LIN {X 0,Y 192.714,Z 301.29,A -85,B 0,C 180,E1 -21855.206,E2 -21855.206} C_VEL
LIN {X 0,Y 192.91,Z 301.267,A -85,B 0,C 180,E1 -21859.549,E2 -21859.549} C_VEL
LIN {X 0,Y 193.003,Z 301.257,A -85,B 0,C 180,E1 -21861.621,E2 -21861.621} C_VEL
LIN {X 0,Y 193.24,Z 301.226,A -85,B 0,C 180,E1 -21867.912,E2 -21867.912} C_VEL
LIN {X 0,Y 193.401,Z 301.208,A -85,B 0,C 180,E1 -21869.996,E2 -21869.996} C_VEL
LIN {X 0,Y 192.941,Z 301.26,A -85,B 0,C 180,E1 -21874.174,E2 -21874.174} C_VEL
LIN {X 0,Y 193,Z 301.258,A -85,B 0,C 180,E1 -21878.372,E2 -21878.372} C_VEL
LIN {X 0,Y 192.755,Z 301.282,A -85,B 0,C 180,E1 -21882.633,E2 -21882.633} C_VEL
LIN {X 0,Y 192.704,Z 301.293,A -85,B 0,C 180,E1 -21886.96,E2 -21886.96} C_VEL
LIN {X 0,Y 192.567,Z 301.305,A -85,B 0,C 180,E1 -21891.401,E2 -21891.401} C_VEL
LIN {X 0,Y 192.6,Z 301.303,A -85,B 0,C 180,E1 -21894.214,E2 -21894.214} C_VEL
LIN {X 0,Y 192.604,Z 301.305,A -85,B 0,C 180,E1 -21898.895,E2 -21898.895} C_VEL
LIN {X 0,Y 192.556,Z 301.311,A -85,B 0,C 180,E1 -21903.189,E2 -21903.189} C_VEL
LIN {X 0,Y 192.57,Z 301.307,A -85,B 0,C 180,E1 -21908.342,E2 -21908.342} C_VEL
LIN {X 0,Y 192.587,Z 301.308,A -85,B 0,C 180,E1 -21913.145,E2 -21913.145} C_VEL
LIN {X 0,Y 192.582,Z 301.308,A -85,B 0,C 180,E1 -21916.869,E2 -21916.869} C_VEL
LIN {X 0,Y 192.564,Z 301.311,A -85,B 0,C 180,E1 -21921.667,E2 -21921.667} C_VEL
LIN {X 0,Y 192.564,Z 301.308,A -85,B 0,C 180,E1 -21926.822,E2 -21926.822} C_VEL
LIN {X 0,Y 192.629,Z 301.303,A -85,B 0,C 180,E1 -21931.7,E2 -21931.7} C_VEL
LIN {X 0,Y 192.655,Z 301.295,A -85,B 0,C 180,E1 -21936.355,E2 -21936.355} C_VEL
LIN {X 0,Y 192.672,Z 301.296,A -85,B 0,C 180,E1 -21941.498,E2 -21941.498} C_VEL
LIN {X 0,Y 192.716,Z 301.288,A -85,B 0,C 180,E1 -21945.222,E2 -21945.222} C_VEL
LIN {X 0,Y 192.925,Z 301.264,A -85,B 0,C 180,E1 -21949.577,E2 -21949.577} C_VEL
LIN {X 0,Y 192.954,Z 301.26,A -85,B 0,C 180,E1 -21953.738,E2 -21953.738} C_VEL
LIN {X 0,Y 193.218,Z 301.227,A -85,B 0,C 180,E1 -21957.926,E2 -21957.926} C_VEL
LIN {X 0,Y 193.4,Z 301.206,A -85,B 0,C 180,E1 -21960.01,E2 -21960.01} C_VEL
LIN {X 0,Y 192.932,Z 301.261,A -85,B 0,C 180,E1 -21964.188,E2 -21964.188} C_VEL
LIN {X 0,Y 193.012,Z 301.254,A -85,B 0,C 180,E1 -21968.385,E2 -21968.385} C_VEL
LIN {X 0,Y 192.769,Z 301.283,A -85,B 0,C 180,E1 -21972.646,E2 -21972.646} C_VEL
LIN {X 0,Y 192.691,Z 301.294,A -85,B 0,C 180,E1 -21978.518,E2 -21978.518} C_VEL
LIN {X 0,Y 192.61,Z 301.301,A -85,B 0,C 180,E1 -21984.198,E2 -21984.198} C_VEL
LIN {X 0,Y 192.602,Z 301.305,A -85,B 0,C 180,E1 -21988.874,E2 -21988.874} C_VEL
LIN {X 0,Y 192.598,Z 301.304,A -85,B 0,C 180,E1 -21993.196,E2 -21993.196} C_VEL
LIN {X 0,Y 192.547,Z 301.31,A -85,B 0,C 180,E1 -21998.364,E2 -21998.364} C_VEL
LIN {X 0,Y 192.492,Z 301.317,A -85,B 0,C 180,E1 -22003.102,E2 -22003.102} C_VEL
LIN {X 0,Y 192.493,Z 301.317,A -85,B 0,C 180,E1 -22006.916,E2 -22006.916} C_VEL
LIN {X 0,Y 192.553,Z 301.31,A -85,B 0,C 180,E1 -22011.654,E2 -22011.654} C_VEL
LIN {X 0,Y 192.608,Z 301.301,A -85,B 0,C 180,E1 -22016.821,E2 -22016.821} C_VEL
LIN {X 0,Y 192.73,Z 301.288,A -85,B 0,C 180,E1 -22021.707,E2 -22021.707} C_VEL
LIN {X 0,Y 193.398,Z 301.317,A -85,B 0,C 180,E1 -22026.256,E2 -22026.256} C_VEL
LIN {X 0,Y 192.681,Z 306.854,A -85,B 0,C 180,E1 -22029.172,E2 -22029.172} C_VEL
LIN {X 0,Y 192.12,Z 311.73,A -85,B 0,C 180,E1 -22031.771,E2 -22031.771} C_VEL
LIN {X 0,Y 192.839,Z 333.39,A -85,B 0,C 180,E1 -22033.223,E2 -22033.223} C_VEL
LIN {X 0,Y 194.563,Z 352.743,A -85,B 0,C 180,E1 -22034.487,E2 -22034.487} C_VEL
LIN {X 0,Y 193.91,Z 391.128,A -85,B 0,C 180,E1 -22037.244,E2 -22037.244} C_VEL
LIN {X 0,Y 193.573,Z 403.683,A -85,B 0,C 180,E1 -22038.585,E2 -22038.585} C_VEL
LIN {X 0,Y 193.177,Z 413.704,A -85,B 0,C 180,E1 -22040.036,E2 -22040.036} C_VEL
LIN {X 0,Y 192.88,Z 423.653,A -85,B 0,C 180,E1 -22041.84,E2 -22041.84} C_VEL
LIN {X 0,Y 192.134,Z 428.371,A -85,B 0,C 180,E1 -22042.875,E2 -22042.875} C_VEL
LIN {X 0,Y 190.518,Z 432.587,A -85,B 0,C 180,E1 -22044.037,E2 -22044.037} C_VEL
LIN {X 0,Y 186.361,Z 441.213,A -85,B 0,C 180,E1 -22047.161,E2 -22047.161} C_VEL
LIN {X 0,Y 185.667,Z 444.803,A -85,B 0,C 180,E1 -22048.63,E2 -22048.63} C_VEL
LIN {X 0,Y 185.446,Z 450.471,A -85,B 0,C 180,E1 -22051.089,E2 -22051.089} C_VEL
LIN {X 0,Y 184.916,Z 454.487,A -85,B 0,C 180,E1 -22053.272,E2 -22053.272} C_VEL
LIN {X 0,Y 184.491,Z 459.134,A -85,B 0,C 180,E1 -22056.566,E2 -22056.566} C_VEL
LIN {X 0,Y 184.526,Z 461.668,A -85,B 0,C 180,E1 -22058.767,E2 -22058.767} C_VEL
LIN {X 0,Y 184.887,Z 463.625,A -85,B 0,C 180,E1 -22060.96,E2 -22060.96} C_VEL
LIN {X 0,Y 186.868,Z 466.287,A -85,B 0,C 180,E1 -22065.267,E2 -22065.267} C_VEL
LIN {X 0,Y 188.38,Z 466.993,A -85,B 0,C 180,E1 -22067.369,E2 -22067.369} C_VEL
LIN {X 0,Y 192.458,Z 467.07,A -85,B 0,C 180,E1 -22071.422,E2 -22071.422} C_VEL
LIN {X 0,Y 194.9,Z 466.532,A -85,B 0,C 180,E1 -22073.373,E2 -22073.373} C_VEL
LIN {X 0,Y 201.021,Z 463.983,A -85,B 0,C 180,E1 -22077.036,E2 -22077.036} C_VEL
LIN {X 0,Y 206.371,Z 460.911,A -85,B 0,C 180,E1 -22079.594,E2 -22079.594} C_VEL
LIN {X 0,Y 212.35,Z 456.67,A -85,B 0,C 180,E1 -22081.978,E2 -22081.978} C_VEL
LIN {X 0,Y 218.89,Z 451.233,A -85,B 0,C 180,E1 -22084.189,E2 -22084.189} C_VEL
LIN {X 0,Y 225.921,Z 444.175,A -85,B 0,C 180,E1 -22086.235,E2 -22086.235} C_VEL
LIN {X 0,Y 232.58,Z 436.469,A -85,B 0,C 180,E1 -22087.893,E2 -22087.893} C_VEL
LIN {X 0,Y 238.884,Z 428.028,A -85,B 0,C 180,E1 -22089.24,E2 -22089.24} C_VEL
LIN {X 0,Y 245.835,Z 416.876,A -85,B 0,C 180,E1 -22090.573,E2 -22090.573} C_VEL
LIN {X 0,Y 250.951,Z 407.114,A -85,B 0,C 180,E1 -22091.427,E2 -22091.427} C_VEL
LIN {X 0,Y 256.021,Z 395.266,A -85,B 0,C 180,E1 -22092.232,E2 -22092.232} C_VEL
LIN {X 0,Y 256.411,Z 394.123,A -85,B 0,C 180,E1 -22092.301,E2 -22092.301} C_VEL
LIN {X 0,Y 256.828,Z 392.188,A -85,B 0,C 180,E1 -22092.829,E2 -22092.829} C_VEL
LIN {X 0,Y 256.986,Z 390.311,A -85,B 0,C 180,E1 -22094.672,E2 -22094.672} C_VEL
LIN {X 0,Y 257.234,Z 390.123,A -85,B 0,C 180,E1 -22097.537,E2 -22097.537} C_VEL
LIN {X 0,Y 256.903,Z 391.834,A -85,B 0,C 180,E1 -22098.331,E2 -22098.331} C_VEL
LIN {X 0,Y 252.117,Z 403.433,A -85,B 0,C 180,E1 -22099.207,E2 -22099.207} C_VEL
LIN {X 0,Y 246.872,Z 413.507,A -85,B 0,C 180,E1 -22100.235,E2 -22100.235} C_VEL
LIN {X 0,Y 240.553,Z 423.709,A -85,B 0,C 180,E1 -22101.614,E2 -22101.614} C_VEL
LIN {X 0,Y 234.297,Z 432.009,A -85,B 0,C 180,E1 -22103.127,E2 -22103.127} C_VEL
LIN {X 0,Y 228.3,Z 438.772,A -85,B 0,C 180,E1 -22104.738,E2 -22104.738} C_VEL
LIN {X 0,Y 222.538,Z 444.44,A -85,B 0,C 180,E1 -22106.441,E2 -22106.441} C_VEL
LIN {X 0,Y 216.108,Z 449.749,A -85,B 0,C 180,E1 -22108.637,E2 -22108.637} C_VEL
LIN {X 0,Y 210.136,Z 453.681,A -85,B 0,C 180,E1 -22110.981,E2 -22110.981} C_VEL
LIN {X 0,Y 204.689,Z 456.441,A -85,B 0,C 180,E1 -22113.481,E2 -22113.481} C_VEL
LIN {X 0,Y 200.615,Z 457.914,A -85,B 0,C 180,E1 -22115.628,E2 -22115.628} C_VEL
LIN {X 0,Y 198.22,Z 458.508,A -85,B 0,C 180,E1 -22117.035,E2 -22117.035} C_VEL
LIN {X 0,Y 192.832,Z 458.677,A -85,B 0,C 180,E1 -22120.842,E2 -22120.842} C_VEL
LIN {X 0,Y 190.607,Z 458.14,A -85,B 0,C 180,E1 -22122.834,E2 -22122.834} C_VEL
LIN {X 0,Y 188.84,Z 457.038,A -85,B 0,C 180,E1 -22124.889,E2 -22124.889} C_VEL
LIN {X 0,Y 187.164,Z 455.517,A -85,B 0,C 180,E1 -22126.969,E2 -22126.969} C_VEL
LIN {X 0,Y 185.254,Z 451.978,A -85,B 0,C 180,E1 -22130.545,E2 -22130.545} C_VEL
LIN {X 0,Y 184.338,Z 446.507,A -85,B 0,C 180,E1 -22134.52,E2 -22134.52} C_VEL
LIN {X 0,Y 184.067,Z 440.418,A -85,B 0,C 180,E1 -22137.801,E2 -22137.801} C_VEL
LIN {X 0,Y 184.266,Z 434.187,A -85,B 0,C 180,E1 -22140.535,E2 -22140.535} C_VEL
LIN {X 0,Y 184.542,Z 428.076,A -85,B 0,C 180,E1 -22142.717,E2 -22142.717} C_VEL
LIN {X 0,Y 184.867,Z 418.775,A -85,B 0,C 180,E1 -22145.442,E2 -22145.442} C_VEL
LIN {X 0,Y 185.395,Z 408.039,A -85,B 0,C 180,E1 -22147.887,E2 -22147.887} C_VEL
LIN {X 0,Y 185.843,Z 397.669,A -85,B 0,C 180,E1 -22149.761,E2 -22149.761} C_VEL
LIN {X 0,Y 186.323,Z 385.441,A -85,B 0,C 180,E1 -22151.442,E2 -22151.442} C_VEL
LIN {X 0,Y 186.787,Z 373.89,A -85,B 0,C 180,E1 -22152.579,E2 -22152.579} C_VEL
LIN {X 0,Y 187.665,Z 320.595,A -85,B 0,C 180,E1 -22156.44,E2 -22156.44} C_VEL
LIN {X 0,Y 185.761,Z 302.162,A -85,B 0,C 180,E1 -22157.692,E2 -22157.692} C_VEL
LIN {X 0,Y 185.579,Z 302.177,A -85,B 0,C 180,E1 -22162.24,E2 -22162.24} C_VEL
LIN {X 0,Y 185.493,Z 302.19,A -85,B 0,C 180,E1 -22167.029,E2 -22167.029} C_VEL
LIN {X 0,Y 185.532,Z 302.184,A -85,B 0,C 180,E1 -22169.487,E2 -22169.487} C_VEL
LIN {X 0,Y 185.48,Z 302.194,A -85,B 0,C 180,E1 -22174.621,E2 -22174.621} C_VEL
LIN {X 0,Y 185.481,Z 302.191,A -85,B 0,C 180,E1 -22177.303,E2 -22177.303} C_VEL
LIN {X 0,Y 185.439,Z 302.194,A -85,B 0,C 180,E1 -22180.709,E2 -22180.709} C_VEL
LIN {X 0,Y 185.432,Z 302.198,A -85,B 0,C 180,E1 -22186.045,E2 -22186.045} C_VEL
LIN {X 0,Y 185.43,Z 302.193,A -85,B 0,C 180,E1 -22189.881,E2 -22189.881} C_VEL
LIN {X 0,Y 185.472,Z 302.193,A -85,B 0,C 180,E1 -22192.703,E2 -22192.703} C_VEL
LIN {X 0,Y 185.501,Z 302.184,A -85,B 0,C 180,E1 -22197.963,E2 -22197.963} C_VEL
LIN {X 0,Y 185.518,Z 302.189,A -85,B 0,C 180,E1 -22202.957,E2 -22202.957} C_VEL
LIN {X 0,Y 185.538,Z 302.182,A -85,B 0,C 180,E1 -22207.738,E2 -22207.738} C_VEL
LIN {X 0,Y 185.646,Z 302.171,A -85,B 0,C 180,E1 -22212.367,E2 -22212.367} C_VEL
LIN {X 0,Y 185.685,Z 302.161,A -85,B 0,C 180,E1 -22216.87,E2 -22216.87} C_VEL
LIN {X 0,Y 185.949,Z 302.134,A -85,B 0,C 180,E1 -22221.301,E2 -22221.301} C_VEL
LIN {X 0,Y 186.182,Z 302.104,A -85,B 0,C 180,E1 -22227.833,E2 -22227.833} C_VEL
LIN {X 0,Y 186.365,Z 302.085,A -85,B 0,C 180,E1 -22229.996,E2 -22229.996} C_VEL
LIN {X 0,Y 185.887,Z 302.138,A -85,B 0,C 180,E1 -22234.333,E2 -22234.333} C_VEL
LIN {X 0,Y 185.945,Z 302.135,A -85,B 0,C 180,E1 -22238.692,E2 -22238.692} C_VEL
LIN {X 0,Y 185.68,Z 302.161,A -85,B 0,C 180,E1 -22243.122,E2 -22243.122} C_VEL
LIN {X 0,Y 185.639,Z 302.172,A -85,B 0,C 180,E1 -22247.626,E2 -22247.626} C_VEL
LIN {X 0,Y 185.529,Z 302.183,A -85,B 0,C 180,E1 -22252.256,E2 -22252.256} C_VEL
LIN {X 0,Y 185.514,Z 302.189,A -85,B 0,C 180,E1 -22257.035,E2 -22257.035} C_VEL
LIN {X 0,Y 185.534,Z 302.183,A -85,B 0,C 180,E1 -22259.496,E2 -22259.496} C_VEL
LIN {X 0,Y 185.477,Z 302.192,A -85,B 0,C 180,E1 -22264.632,E2 -22264.632} C_VEL
LIN {X 0,Y 185.526,Z 302.187,A -85,B 0,C 180,E1 -22267.319,E2 -22267.319} C_VEL
LIN {X 0,Y 185.541,Z 302.181,A -85,B 0,C 180,E1 -22270.77,E2 -22270.77} C_VEL
LIN {X 0,Y 185.543,Z 302.184,A -85,B 0,C 180,E1 -22276.022,E2 -22276.022} C_VEL
LIN {X 0,Y 185.508,Z 302.185,A -85,B 0,C 180,E1 -22279.923,E2 -22279.923} C_VEL
LIN {X 0,Y 185.524,Z 302.186,A -85,B 0,C 180,E1 -22282.707,E2 -22282.707} C_VEL
LIN {X 0,Y 185.507,Z 302.184,A -85,B 0,C 180,E1 -22287.983,E2 -22287.983} C_VEL
LIN {X 0,Y 185.549,Z 302.182,A -85,B 0,C 180,E1 -22290.586,E2 -22290.586} C_VEL
LIN {X 0,Y 185.551,Z 302.183,A -85,B 0,C 180,E1 -22295.391,E2 -22295.391} C_VEL
LIN {X 0,Y 185.607,Z 302.176,A -85,B 0,C 180,E1 -22301.181,E2 -22301.181} C_VEL
LIN {X 0,Y 185.645,Z 302.169,A -85,B 0,C 180,E1 -22304.645,E2 -22304.645} C_VEL
LIN {X 0,Y 185.868,Z 302.143,A -85,B 0,C 180,E1 -22309.429,E2 -22309.429} C_VEL
LIN {X 0,Y 185.918,Z 302.136,A -85,B 0,C 180,E1 -22313.5,E2 -22313.5} C_VEL
LIN {X 0,Y 186.164,Z 302.105,A -85,B 0,C 180,E1 -22317.847,E2 -22317.847} C_VEL
LIN {X 0,Y 186.366,Z 302.082,A -85,B 0,C 180,E1 -22320.011,E2 -22320.011} C_VEL
LIN {X 0,Y 185.88,Z 302.139,A -85,B 0,C 180,E1 -22324.347,E2 -22324.347} C_VEL
LIN {X 0,Y 185.963,Z 302.134,A -85,B 0,C 180,E1 -22328.705,E2 -22328.705} C_VEL
LIN {X 0,Y 185.693,Z 302.162,A -85,B 0,C 180,E1 -22333.136,E2 -22333.136} C_VEL
LIN {X 0,Y 185.621,Z 302.176,A -85,B 0,C 180,E1 -22338.831,E2 -22338.831} C_VEL
LIN {X 0,Y 185.544,Z 302.182,A -85,B 0,C 180,E1 -22344.634,E2 -22344.634} C_VEL
LIN {X 0,Y 185.546,Z 302.183,A -85,B 0,C 180,E1 -22349.51,E2 -22349.51} C_VEL
LIN {X 0,Y 185.501,Z 302.188,A -85,B 0,C 180,E1 -22354.643,E2 -22354.643} C_VEL
LIN {X 0,Y 185.506,Z 302.191,A -85,B 0,C 180,E1 -22357.324,E2 -22357.324} C_VEL
LIN {X 0,Y 185.468,Z 302.188,A -85,B 0,C 180,E1 -22360.73,E2 -22360.73} C_VEL
LIN {X 0,Y 185.464,Z 302.195,A -85,B 0,C 180,E1 -22366.066,E2 -22366.066} C_VEL
LIN {X 0,Y 185.466,Z 302.191,A -85,B 0,C 180,E1 -22369.9,E2 -22369.9} C_VEL
LIN {X 0,Y 185.513,Z 302.187,A -85,B 0,C 180,E1 -22372.722,E2 -22372.722} C_VEL
LIN {X 0,Y 185.556,Z 302.18,A -85,B 0,C 180,E1 -22377.982,E2 -22377.982} C_VEL
LIN {X 0,Y 186.194,Z 302.106,A -85,B 0,C 180,E1 -22385.472,E2 -22385.472} C_VEL
LIN {X 0,Y 186.297,Z 302.281,A -85,B 0,C 180,E1 -22386.816,E2 -22386.816} C_VEL
LIN {X 0,Y 185.057,Z 311.759,A -85,B 0,C 180,E1 -22391.944,E2 -22391.944} C_VEL
LIN {X 0,Y 185.765,Z 333.185,A -85,B 0,C 180,E1 -22393.45,E2 -22393.45} C_VEL
LIN {X 0,Y 187.497,Z 353.905,A -85,B 0,C 180,E1 -22394.862,E2 -22394.862} C_VEL
LIN {X 0,Y 186.922,Z 391.639,A -85,B 0,C 180,E1 -22397.711,E2 -22397.711} C_VEL
LIN {X 0,Y 186.629,Z 403.007,A -85,B 0,C 180,E1 -22398.985,E2 -22398.985} C_VEL
LIN {X 0,Y 186.293,Z 412.343,A -85,B 0,C 180,E1 -22400.368,E2 -22400.368} C_VEL
LIN {X 0,Y 186.051,Z 420.491,A -85,B 0,C 180,E1 -22401.86,E2 -22401.86} C_VEL
LIN {X 0,Y 185.911,Z 429.013,A -85,B 0,C 180,E1 -22403.764,E2 -22403.764} C_VEL
LIN {X 0,Y 185.786,Z 437.878,A -85,B 0,C 180,E1 -22406.208,E2 -22406.208} C_VEL
LIN {X 0,Y 185.667,Z 444.803,A -85,B 0,C 180,E1 -22408.63,E2 -22408.63} C_VEL
LIN {X 0,Y 184.87,Z 448.155,A -85,B 0,C 180,E1 -22410.123,E2 -22410.123} C_VEL
LIN {X 0,Y 183.078,Z 450.876,A -85,B 0,C 180,E1 -22411.673,E2 -22411.673} C_VEL
LIN {X 0,Y 178.945,Z 455.26,A -85,B 0,C 180,E1 -22414.984,E2 -22414.984} C_VEL
LIN {X 0,Y 177.782,Z 457.288,A -85,B 0,C 180,E1 -22416.77,E2 -22416.77} C_VEL
LIN {X 0,Y 177.682,Z 457.975,A -85,B 0,C 180,E1 -22417.378,E2 -22417.378} C_VEL
LIN {X 0,Y 178.095,Z 462.105,A -85,B 0,C 180,E1 -22421.383,E2 -22421.383} C_VEL
LIN {X 0,Y 178.874,Z 463.941,A -85,B 0,C 180,E1 -22423.639,E2 -22423.639} C_VEL
LIN {X 0,Y 180.092,Z 465.258,A -85,B 0,C 180,E1 -22425.857,E2 -22425.857} C_VEL
LIN {X 0,Y 183.564,Z 466.716,A -85,B 0,C 180,E1 -22430.16,E2 -22430.16} C_VEL
LIN {X 0,Y 185.866,Z 466.807,A -85,B 0,C 180,E1 -22432.221,E2 -22432.221} C_VEL
LIN {X 0,Y 188.41,Z 466.444,A -85,B 0,C 180,E1 -22434.228,E2 -22434.228} C_VEL
LIN {X 0,Y 191.417,Z 465.754,A -85,B 0,C 180,E1 -22436.145,E2 -22436.145} C_VEL
LIN {X 0,Y 194.745,Z 464.612,A -85,B 0,C 180,E1 -22437.982,E2 -22437.982} C_VEL
LIN {X 0,Y 200.286,Z 462.013,A -85,B 0,C 180,E1 -22440.588,E2 -22440.588} C_VEL
LIN {X 0,Y 206.467,Z 458.338,A -85,B 0,C 180,E1 -22443.003,E2 -22443.003} C_VEL
LIN {X 0,Y 213.171,Z 453.38,A -85,B 0,C 180,E1 -22445.24,E2 -22445.24} C_VEL
LIN {X 0,Y 219.155,Z 448.297,A -85,B 0,C 180,E1 -22446.965,E2 -22446.965} C_VEL
LIN {X 0,Y 225.522,Z 442.056,A -85,B 0,C 180,E1 -22448.558,E2 -22448.558} C_VEL
LIN {X 0,Y 230.87,Z 436.054,A -85,B 0,C 180,E1 -22449.74,E2 -22449.74} C_VEL
LIN {X 0,Y 236.469,Z 429.072,A -85,B 0,C 180,E1 -22450.836,E2 -22450.836} C_VEL
LIN {X 0,Y 242.968,Z 419.627,A -85,B 0,C 180,E1 -22451.986,E2 -22451.986} C_VEL
LIN {X 0,Y 249.315,Z 408.307,A -85,B 0,C 180,E1 -22452.985,E2 -22452.985} C_VEL
LIN {X 0,Y 254.166,Z 397.922,A -85,B 0,C 180,E1 -22453.735,E2 -22453.735} C_VEL
LIN {X 0,Y 254.39,Z 396.608,A -85,B 0,C 180,E1 -22455.917,E2 -22455.917} C_VEL
LIN {X 0,Y 254.529,Z 396.583,A -85,B 0,C 180,E1 -22456.978,E2 -22456.978} C_VEL
LIN {X 0,Y 249.745,Z 406.704,A -85,B 0,C 180,E1 -22457.821,E2 -22457.821} C_VEL
LIN {X 0,Y 243.869,Z 417.129,A -85,B 0,C 180,E1 -22458.915,E2 -22458.915} C_VEL
LIN {X 0,Y 237.777,Z 425.871,A -85,B 0,C 180,E1 -22460.137,E2 -22460.137} C_VEL
LIN {X 0,Y 231.605,Z 433.4,A -85,B 0,C 180,E1 -22461.524,E2 -22461.524} C_VEL
LIN {X 0,Y 225.335,Z 440.075,A -85,B 0,C 180,E1 -22463.093,E2 -22463.093} C_VEL
LIN {X 0,Y 219.316,Z 445.481,A -85,B 0,C 180,E1 -22464.764,E2 -22464.764} C_VEL
LIN {X 0,Y 212.46,Z 450.613,A -85,B 0,C 180,E1 -22466.911,E2 -22466.911} C_VEL
LIN {X 0,Y 206.113,Z 454.397,A -85,B 0,C 180,E1 -22469.229,E2 -22469.229} C_VEL
LIN {X 0,Y 202.151,Z 456.338,A -85,B 0,C 180,E1 -22470.865,E2 -22470.865} C_VEL
LIN {X 0,Y 198.46,Z 457.731,A -85,B 0,C 180,E1 -22472.58,E2 -22472.58} C_VEL
LIN {X 0,Y 194.235,Z 458.809,A -85,B 0,C 180,E1 -22474.772,E2 -22474.772} C_VEL
LIN {X 0,Y 188.838,Z 459.247,A -85,B 0,C 180,E1 -22478.14,E2 -22478.14} C_VEL
LIN {X 0,Y 186.159,Z 458.779,A -85,B 0,C 180,E1 -22480.127,E2 -22480.127} C_VEL
LIN {X 0,Y 183.84,Z 457.91,A -85,B 0,C 180,E1 -22482.181,E2 -22482.181} C_VEL
LIN {X 0,Y 182.018,Z 456.683,A -85,B 0,C 180,E1 -22484.308,E2 -22484.308} C_VEL
LIN {X 0,Y 179.584,Z 453.835,A -85,B 0,C 180,E1 -22487.56,E2 -22487.56} C_VEL
LIN {X 0,Y 178.124,Z 449.933,A -85,B 0,C 180,E1 -22490.909,E2 -22490.909} C_VEL
LIN {X 0,Y 177.443,Z 444.913,A -85,B 0,C 180,E1 -22494.306,E2 -22494.306} C_VEL
LIN {X 0,Y 177.217,Z 438.44,A -85,B 0,C 180,E1 -22497.716,E2 -22497.716} C_VEL
LIN {X 0,Y 177.549,Z 430.204,A -85,B 0,C 180,E1 -22501.123,E2 -22501.123} C_VEL
LIN {X 0,Y 177.738,Z 423.377,A -85,B 0,C 180,E1 -22503.389,E2 -22503.389} C_VEL
LIN {X 0,Y 178.126,Z 415.112,A -85,B 0,C 180,E1 -22505.649,E2 -22505.649} C_VEL
LIN {X 0,Y 178.522,Z 406.284,A -85,B 0,C 180,E1 -22507.623,E2 -22507.623} C_VEL
LIN {X 0,Y 179.031,Z 393.922,A -85,B 0,C 180,E1 -22509.786,E2 -22509.786} C_VEL
LIN {X 0,Y 179.432,Z 383.508,A -85,B 0,C 180,E1 -22511.162,E2 -22511.162} C_VEL
LIN {X 0,Y 179.823,Z 371.216,A -85,B 0,C 180,E1 -22512.369,E2 -22512.369} C_VEL
LIN {X 0,Y 180.63,Z 321.144,A -85,B 0,C 180,E1 -22516.191,E2 -22516.191} C_VEL
LIN {X 0,Y 178.718,Z 303.039,A -85,B 0,C 180,E1 -22517.509,E2 -22517.509} C_VEL
LIN {X 0,Y 178.494,Z 303.057,A -85,B 0,C 180,E1 -22523.174,E2 -22523.174} C_VEL
LIN {X 0,Y 178.43,Z 303.072,A -85,B 0,C 180,E1 -22528.192,E2 -22528.192} C_VEL
LIN {X 0,Y 178.468,Z 303.063,A -85,B 0,C 180,E1 -22533.441,E2 -22533.441} C_VEL
LIN {X 0,Y 178.367,Z 303.075,A -85,B 0,C 180,E1 -22539.065,E2 -22539.065} C_VEL
LIN {X 0,Y 178.371,Z 303.074,A -85,B 0,C 180,E1 -22542.035,E2 -22542.035} C_VEL
LIN {X 0,Y 178.368,Z 303.079,A -85,B 0,C 180,E1 -22545.153,E2 -22545.153} C_VEL
LIN {X 0,Y 178.372,Z 303.076,A -85,B 0,C 180,E1 -22548.45,E2 -22548.45} C_VEL
LIN {X 0,Y 178.389,Z 303.075,A -85,B 0,C 180,E1 -22553.771,E2 -22553.771} C_VEL
LIN {X 0,Y 178.452,Z 303.067,A -85,B 0,C 180,E1 -22556.535,E2 -22556.535} C_VEL
LIN {X 0,Y 178.435,Z 303.07,A -85,B 0,C 180,E1 -22561.79,E2 -22561.79} C_VEL
LIN {X 0,Y 178.458,Z 303.064,A -85,B 0,C 180,E1 -22566.804,E2 -22566.804} C_VEL
LIN {X 0,Y 178.608,Z 303.05,A -85,B 0,C 180,E1 -22571.648,E2 -22571.648} C_VEL
LIN {X 0,Y 178.613,Z 303.042,A -85,B 0,C 180,E1 -22576.341,E2 -22576.341} C_VEL
LIN {X 0,Y 178.881,Z 303.014,A -85,B 0,C 180,E1 -22580.954,E2 -22580.954} C_VEL
LIN {X 0,Y 179.125,Z 302.983,A -85,B 0,C 180,E1 -22587.748,E2 -22587.748} C_VEL
LIN {X 0,Y 179.329,Z 302.961,A -85,B 0,C 180,E1 -22589.996,E2 -22589.996} C_VEL
LIN {X 0,Y 178.833,Z 303.016,A -85,B 0,C 180,E1 -22594.504,E2 -22594.504} C_VEL
LIN {X 0,Y 178.877,Z 303.014,A -85,B 0,C 180,E1 -22599.038,E2 -22599.038} C_VEL
LIN {X 0,Y 178.608,Z 303.042,A -85,B 0,C 180,E1 -22603.652,E2 -22603.652} C_VEL
LIN {X 0,Y 178.574,Z 303.052,A -85,B 0,C 180,E1 -22609.214,E2 -22609.214} C_VEL
LIN {X 0,Y 178.474,Z 303.065,A -85,B 0,C 180,E1 -22615.116,E2 -22615.116} C_VEL
LIN {X 0,Y 178.478,Z 303.062,A -85,B 0,C 180,E1 -22619.997,E2 -22619.997} C_VEL
LIN {X 0,Y 178.441,Z 303.068,A -85,B 0,C 180,E1 -22624.223,E2 -22624.223} C_VEL
LIN {X 0,Y 178.444,Z 303.067,A -85,B 0,C 180,E1 -22629.056,E2 -22629.056} C_VEL
LIN {X 0,Y 178.473,Z 303.062,A -85,B 0,C 180,E1 -22632.017,E2 -22632.017} C_VEL
LIN {X 0,Y 178.489,Z 303.065,A -85,B 0,C 180,E1 -22635.127,E2 -22635.127} C_VEL
LIN {X 0,Y 178.47,Z 303.062,A -85,B 0,C 180,E1 -22638.428,E2 -22638.428} C_VEL
LIN {X 0,Y 178.423,Z 303.072,A -85,B 0,C 180,E1 -22643.8,E2 -22643.8} C_VEL
LIN {X 0,Y 178.455,Z 303.065,A -85,B 0,C 180,E1 -22646.556,E2 -22646.556} C_VEL
LIN {X 0,Y 178.489,Z 303.062,A -85,B 0,C 180,E1 -22650.016,E2 -22650.016} C_VEL
LIN {X 0,Y 178.49,Z 303.061,A -85,B 0,C 180,E1 -22654.896,E2 -22654.896} C_VEL
LIN {X 0,Y 178.564,Z 303.053,A -85,B 0,C 180,E1 -22660.825,E2 -22660.825} C_VEL
LIN {X 0,Y 178.621,Z 303.043,A -85,B 0,C 180,E1 -22666.357,E2 -22666.357} C_VEL
LIN {X 0,Y 178.889,Z 303.013,A -85,B 0,C 180,E1 -22670.971,E2 -22670.971} C_VEL
LIN {X 0,Y 179.112,Z 302.983,A -85,B 0,C 180,E1 -22677.763,E2 -22677.763} C_VEL
LIN {X 0,Y 179.331,Z 302.958,A -85,B 0,C 180,E1 -22680.011,E2 -22680.011} C_VEL
LIN {X 0,Y 178.829,Z 303.017,A -85,B 0,C 180,E1 -22684.519,E2 -22684.519} C_VEL
LIN {X 0,Y 178.894,Z 303.014,A -85,B 0,C 180,E1 -22689.052,E2 -22689.052} C_VEL
LIN {X 0,Y 178.62,Z 303.041,A -85,B 0,C 180,E1 -22693.666,E2 -22693.666} C_VEL
LIN {X 0,Y 178.551,Z 303.056,A -85,B 0,C 180,E1 -22699.163,E2 -22699.163} C_VEL
LIN {X 0,Y 178.465,Z 303.066,A -85,B 0,C 180,E1 -22705.087,E2 -22705.087} C_VEL
LIN {X 0,Y 178.463,Z 303.063,A -85,B 0,C 180,E1 -22710.805,E2 -22710.805} C_VEL
LIN {X 0,Y 178.487,Z 303.062,A -85,B 0,C 180,E1 -22714.228,E2 -22714.228} C_VEL
LIN {X 0,Y 178.393,Z 303.073,A -85,B 0,C 180,E1 -22719.087,E2 -22719.087} C_VEL
LIN {X 0,Y 178.401,Z 303.073,A -85,B 0,C 180,E1 -22722.057,E2 -22722.057} C_VEL
LIN {X 0,Y 178.4,Z 303.074,A -85,B 0,C 180,E1 -22725.175,E2 -22725.175} C_VEL
LIN {X 0,Y 178.407,Z 303.069,A -85,B 0,C 180,E1 -22728.471,E2 -22728.471} C_VEL
LIN {X 0,Y 178.432,Z 303.072,A -85,B 0,C 180,E1 -22733.791,E2 -22733.791} C_VEL
LIN {X 0,Y 178.498,Z 303.06,A -85,B 0,C 180,E1 -22736.554,E2 -22736.554} C_VEL
LIN {X 0,Y 178.627,Z 303.046,A -85,B 0,C 180,E1 -22741.832,E2 -22741.832} C_VEL
LIN {X 0,Y 178.984,Z 303.003,A -85,B 0,C 180,E1 -22744.59,E2 -22744.59} C_VEL
LIN {X 0,Y 179.064,Z 303.053,A -85,B 0,C 180,E1 -22747.353,E2 -22747.353} C_VEL
LIN {X 0,Y 178.001,Z 311.381,A -85,B 0,C 180,E1 -22752.112,E2 -22752.112} C_VEL
LIN {X 0,Y 178.735,Z 333.472,A -85,B 0,C 180,E1 -22753.734,E2 -22753.734} C_VEL
LIN {X 0,Y 180.47,Z 354.007,A -85,B 0,C 180,E1 -22755.197,E2 -22755.197} C_VEL
LIN {X 0,Y 180.026,Z 390.324,A -85,B 0,C 180,E1 -22758.074,E2 -22758.074} C_VEL
LIN {X 0,Y 179.766,Z 401.605,A -85,B 0,C 180,E1 -22759.356,E2 -22759.356} C_VEL
LIN {X 0,Y 179.431,Z 412.103,A -85,B 0,C 180,E1 -22760.99,E2 -22760.99} C_VEL
LIN {X 0,Y 179.224,Z 422.199,A -85,B 0,C 180,E1 -22762.965,E2 -22762.965} C_VEL
LIN {X 0,Y 179.038,Z 432.318,A -85,B 0,C 180,E1 -22765.501,E2 -22765.501} C_VEL
LIN {X 0,Y 179.022,Z 439.526,A -85,B 0,C 180,E1 -22767.754,E2 -22767.754} C_VEL
LIN {X 0,Y 178.858,Z 445.385,A -85,B 0,C 180,E1 -22770.004,E2 -22770.004} C_VEL
LIN {X 0,Y 178.494,Z 450.104,A -85,B 0,C 180,E1 -22772.26,E2 -22772.26} C_VEL
LIN {X 0,Y 178.01,Z 454.017,A -85,B 0,C 180,E1 -22774.533,E2 -22774.533} C_VEL
LIN {X 0,Y 177.682,Z 457.975,A -85,B 0,C 180,E1 -22777.378,E2 -22777.378} C_VEL
LIN {X 0,Y 177.105,Z 459.797,A -85,B 0,C 180,E1 -22779.187,E2 -22779.187} C_VEL
LIN {X 0,Y 174.914,Z 461.918,A -85,B 0,C 180,E1 -22782.258,E2 -22782.258} C_VEL
LIN {X 0,Y 173.432,Z 463.603,A -85,B 0,C 180,E1 -22785.436,E2 -22785.436} C_VEL
LIN {X 0,Y 173.954,Z 464.502,A -85,B 0,C 180,E1 -22787.347,E2 -22787.347} C_VEL
LIN {X 0,Y 174.99,Z 465.265,A -85,B 0,C 180,E1 -22788.745,E2 -22788.745} C_VEL
LIN {X 0,Y 179.325,Z 466.319,A -85,B 0,C 180,E1 -22793.077,E2 -22793.077} C_VEL
LIN {X 0,Y 181.969,Z 466.338,A -85,B 0,C 180,E1 -22795.144,E2 -22795.144} C_VEL
LIN {X 0,Y 185.078,Z 465.834,A -85,B 0,C 180,E1 -22797.112,E2 -22797.112} C_VEL
LIN {X 0,Y 192.293,Z 463.697,A -85,B 0,C 180,E1 -22800.779,E2 -22800.779} C_VEL
LIN {X 0,Y 198.419,Z 460.877,A -85,B 0,C 180,E1 -22803.303,E2 -22803.303} C_VEL
LIN {X 0,Y 205.161,Z 456.955,A -85,B 0,C 180,E1 -22805.62,E2 -22805.62} C_VEL
LIN {X 0,Y 212.402,Z 451.852,A -85,B 0,C 180,E1 -22807.747,E2 -22807.747} C_VEL
LIN {X 0,Y 220.177,Z 445.345,A -85,B 0,C 180,E1 -22809.676,E2 -22809.676} C_VEL
LIN {X 0,Y 228.478,Z 437.076,A -85,B 0,C 180,E1 -22811.405,E2 -22811.405} C_VEL
LIN {X 0,Y 234.263,Z 430.265,A -85,B 0,C 180,E1 -22812.458,E2 -22812.458} C_VEL
LIN {X 0,Y 240.975,Z 421.199,A -85,B 0,C 180,E1 -22813.556,E2 -22813.556} C_VEL
LIN {X 0,Y 247.519,Z 410.741,A -85,B 0,C 180,E1 -22814.481,E2 -22814.481} C_VEL
LIN {X 0,Y 250.969,Z 404.101,A -85,B 0,C 180,E1 -22814.947,E2 -22814.947} C_VEL
LIN {X 0,Y 251.331,Z 403.241,A -85,B 0,C 180,E1 -22815.639,E2 -22815.639} C_VEL
LIN {X 0,Y 250.937,Z 404.005,A -85,B 0,C 180,E1 -22815.896,E2 -22815.896} C_VEL
LIN {X 0,Y 245.204,Z 414.192,A -85,B 0,C 180,E1 -22816.811,E2 -22816.811} C_VEL
LIN {X 0,Y 238.671,Z 423.795,A -85,B 0,C 180,E1 -22817.972,E2 -22817.972} C_VEL
LIN {X 0,Y 231.071,Z 432.96,A -85,B 0,C 180,E1 -22819.501,E2 -22819.501} C_VEL
LIN {X 0,Y 225.189,Z 438.964,A -85,B 0,C 180,E1 -22820.794,E2 -22820.794} C_VEL
LIN {X 0,Y 217.484,Z 445.662,A -85,B 0,C 180,E1 -22822.697,E2 -22822.697} C_VEL
LIN {X 0,Y 211.371,Z 450.097,A -85,B 0,C 180,E1 -22824.409,E2 -22824.409} C_VEL
LIN {X 0,Y 204.527,Z 454.125,A -85,B 0,C 180,E1 -22826.637,E2 -22826.637} C_VEL
LIN {X 0,Y 200.181,Z 456.176,A -85,B 0,C 180,E1 -22828.213,E2 -22828.213} C_VEL
LIN {X 0,Y 196.089,Z 457.7,A -85,B 0,C 180,E1 -22829.873,E2 -22829.873} C_VEL
LIN {X 0,Y 192.239,Z 458.806,A -85,B 0,C 180,E1 -22831.613,E2 -22831.613} C_VEL
LIN {X 0,Y 188.251,Z 459.545,A -85,B 0,C 180,E1 -22833.643,E2 -22833.643} C_VEL
LIN {X 0,Y 182.269,Z 459.39,A -85,B 0,C 180,E1 -22837.309,E2 -22837.309} C_VEL
LIN {X 0,Y 179.505,Z 458.766,A -85,B 0,C 180,E1 -22839.357,E2 -22839.357} C_VEL
LIN {X 0,Y 177.113,Z 457.626,A -85,B 0,C 180,E1 -22841.481,E2 -22841.481} C_VEL
LIN {X 0,Y 174.313,Z 455.139,A -85,B 0,C 180,E1 -22844.796,E2 -22844.796} C_VEL
LIN {X 0,Y 172.115,Z 451.616,A -85,B 0,C 180,E1 -22848.208,E2 -22848.208} C_VEL
LIN {X 0,Y 170.873,Z 446.289,A -85,B 0,C 180,E1 -22852.109,E2 -22852.109} C_VEL
LIN {X 0,Y 170.506,Z 440.973,A -85,B 0,C 180,E1 -22855.26,E2 -22855.26} C_VEL
LIN {X 0,Y 170.456,Z 434.847,A -85,B 0,C 180,E1 -22858.216,E2 -22858.216} C_VEL
LIN {X 0,Y 170.796,Z 427.344,A -85,B 0,C 180,E1 -22861.167,E2 -22861.167} C_VEL
LIN {X 0,Y 171.123,Z 417.931,A -85,B 0,C 180,E1 -22864.109,E2 -22864.109} C_VEL
LIN {X 0,Y 171.522,Z 408.463,A -85,B 0,C 180,E1 -22866.458,E2 -22866.458} C_VEL
LIN {X 0,Y 171.808,Z 399.715,A -85,B 0,C 180,E1 -22868.219,E2 -22868.219} C_VEL
LIN {X 0,Y 172.324,Z 388.078,A -85,B 0,C 180,E1 -22870.067,E2 -22870.067} C_VEL
LIN {X 0,Y 172.756,Z 376.24,A -85,B 0,C 180,E1 -22871.414,E2 -22871.414} C_VEL
LIN {X 0,Y 173.639,Z 321.942,A -85,B 0,C 180,E1 -22875.842,E2 -22875.842} C_VEL
LIN {X 0,Y 171.704,Z 303.912,A -85,B 0,C 180,E1 -22877.172,E2 -22877.172} C_VEL
LIN {X 0,Y 171.455,Z 303.937,A -85,B 0,C 180,E1 -22881.635,E2 -22881.635} C_VEL
LIN {X 0,Y 171.379,Z 303.949,A -85,B 0,C 180,E1 -22886.799,E2 -22886.799} C_VEL
LIN {X 0,Y 171.404,Z 303.941,A -85,B 0,C 180,E1 -22890.559,E2 -22890.559} C_VEL
LIN {X 0,Y 171.376,Z 303.949,A -85,B 0,C 180,E1 -22895.022,E2 -22895.022} C_VEL
LIN {X 0,Y 171.323,Z 303.953,A -85,B 0,C 180,E1 -22898.788,E2 -22898.788} C_VEL
LIN {X 0,Y 171.295,Z 303.959,A -85,B 0,C 180,E1 -22904.206,E2 -22904.206} C_VEL
LIN {X 0,Y 171.304,Z 303.954,A -85,B 0,C 180,E1 -22908.968,E2 -22908.968} C_VEL
LIN {X 0,Y 171.331,Z 303.953,A -85,B 0,C 180,E1 -22912.022,E2 -22912.022} C_VEL
LIN {X 0,Y 171.367,Z 303.951,A -85,B 0,C 180,E1 -22915.082,E2 -22915.082} C_VEL
LIN {X 0,Y 171.385,Z 303.945,A -85,B 0,C 180,E1 -22920.518,E2 -22920.518} C_VEL
LIN {X 0,Y 171.408,Z 303.942,A -85,B 0,C 180,E1 -22925.79,E2 -22925.79} C_VEL
LIN {X 0,Y 171.538,Z 303.928,A -85,B 0,C 180,E1 -22930.863,E2 -22930.863} C_VEL
LIN {X 0,Y 171.531,Z 303.926,A -85,B 0,C 180,E1 -22935.765,E2 -22935.765} C_VEL
LIN {X 0,Y 171.819,Z 303.894,A -85,B 0,C 180,E1 -22940.579,E2 -22940.579} C_VEL
LIN {X 0,Y 171.783,Z 303.894,A -85,B 0,C 180,E1 -22945.303,E2 -22945.303} C_VEL
LIN {X 0,Y 172.292,Z 303.838,A -85,B 0,C 180,E1 -22949.996,E2 -22949.996} C_VEL
LIN {X 0,Y 171.781,Z 303.894,A -85,B 0,C 180,E1 -22954.689,E2 -22954.689} C_VEL
LIN {X 0,Y 171.815,Z 303.894,A -85,B 0,C 180,E1 -22959.413,E2 -22959.413} C_VEL
LIN {X 0,Y 171.525,Z 303.926,A -85,B 0,C 180,E1 -22964.227,E2 -22964.227} C_VEL
LIN {X 0,Y 171.493,Z 303.933,A -85,B 0,C 180,E1 -22969.557,E2 -22969.557} C_VEL
LIN {X 0,Y 171.413,Z 303.944,A -85,B 0,C 180,E1 -22975.611,E2 -22975.611} C_VEL
LIN {X 0,Y 171.397,Z 303.944,A -85,B 0,C 180,E1 -22980.59,E2 -22980.59} C_VEL
LIN {X 0,Y 171.365,Z 303.953,A -85,B 0,C 180,E1 -22985.036,E2 -22985.036} C_VEL
LIN {X 0,Y 171.396,Z 303.946,A -85,B 0,C 180,E1 -22988.846,E2 -22988.846} C_VEL
LIN {X 0,Y 171.413,Z 303.944,A -85,B 0,C 180,E1 -22994.181,E2 -22994.181} C_VEL
LIN {X 0,Y 171.387,Z 303.945,A -85,B 0,C 180,E1 -22999.015,E2 -22999.015} C_VEL
LIN {X 0,Y 171.402,Z 303.945,A -85,B 0,C 180,E1 -23002.062,E2 -23002.062} C_VEL
LIN {X 0,Y 171.384,Z 303.944,A -85,B 0,C 180,E1 -23007.801,E2 -23007.801} C_VEL
LIN {X 0,Y 171.415,Z 303.942,A -85,B 0,C 180,E1 -23010.543,E2 -23010.543} C_VEL
LIN {X 0,Y 171.414,Z 303.943,A -85,B 0,C 180,E1 -23015.81,E2 -23015.81} C_VEL
LIN {X 0,Y 171.52,Z 303.93,A -85,B 0,C 180,E1 -23020.878,E2 -23020.878} C_VEL
LIN {X 0,Y 171.535,Z 303.927,A -85,B 0,C 180,E1 -23025.782,E2 -23025.782} C_VEL
LIN {X 0,Y 171.826,Z 303.894,A -85,B 0,C 180,E1 -23030.596,E2 -23030.596} C_VEL
LIN {X 0,Y 171.772,Z 303.893,A -85,B 0,C 180,E1 -23035.318,E2 -23035.318} C_VEL
LIN {X 0,Y 172.296,Z 303.835,A -85,B 0,C 180,E1 -23040.012,E2 -23040.012} C_VEL
LIN {X 0,Y 171.778,Z 303.895,A -85,B 0,C 180,E1 -23044.705,E2 -23044.705} C_VEL
LIN {X 0,Y 171.833,Z 303.892,A -85,B 0,C 180,E1 -23049.427,E2 -23049.427} C_VEL
LIN {X 0,Y 171.535,Z 303.924,A -85,B 0,C 180,E1 -23054.242,E2 -23054.242} C_VEL
LIN {X 0,Y 171.475,Z 303.936,A -85,B 0,C 180,E1 -23059.51,E2 -23059.51} C_VEL
LIN {X 0,Y 171.403,Z 303.946,A -85,B 0,C 180,E1 -23065.581,E2 -23065.581} C_VEL
LIN {X 0,Y 171.42,Z 303.94,A -85,B 0,C 180,E1 -23070.583,E2 -23070.583} C_VEL
LIN {X 0,Y 171.397,Z 303.946,A -85,B 0,C 180,E1 -23075.046,E2 -23075.046} C_VEL
LIN {X 0,Y 171.349,Z 303.95,A -85,B 0,C 180,E1 -23078.811,E2 -23078.811} C_VEL
LIN {X 0,Y 171.327,Z 303.956,A -85,B 0,C 180,E1 -23084.229,E2 -23084.229} C_VEL
LIN {X 0,Y 171.34,Z 303.949,A -85,B 0,C 180,E1 -23088.989,E2 -23088.989} C_VEL
LIN {X 0,Y 171.372,Z 303.95,A -85,B 0,C 180,E1 -23092.043,E2 -23092.043} C_VEL
LIN {X 0,Y 171.412,Z 303.944,A -85,B 0,C 180,E1 -23095.102,E2 -23095.102} C_VEL
LIN {X 0,Y 171.503,Z 303.933,A -85,B 0,C 180,E1 -23100.55,E2 -23100.55} C_VEL
LIN {X 0,Y 171.997,Z 303.875,A -85,B 0,C 180,E1 -23105.887,E2 -23105.887} C_VEL
LIN {X 0,Y 171.748,Z 303.997,A -85,B 0,C 180,E1 -23108.079,E2 -23108.079} C_VEL
LIN {X 0,Y 170.957,Z 310.997,A -85,B 0,C 180,E1 -23112.32,E2 -23112.32} C_VEL
LIN {X 0,Y 171.634,Z 332.542,A -85,B 0,C 180,E1 -23113.997,E2 -23113.997} C_VEL
LIN {X 0,Y 173.482,Z 353.515,A -85,B 0,C 180,E1 -23115.562,E2 -23115.562} C_VEL
LIN {X 0,Y 173.132,Z 390.497,A -85,B 0,C 180,E1 -23118.665,E2 -23118.665} C_VEL
LIN {X 0,Y 172.895,Z 401.962,A -85,B 0,C 180,E1 -23120.056,E2 -23120.056} C_VEL
LIN {X 0,Y 172.602,Z 412.619,A -85,B 0,C 180,E1 -23121.811,E2 -23121.811} C_VEL
LIN {X 0,Y 172.431,Z 422.54,A -85,B 0,C 180,E1 -23123.862,E2 -23123.862} C_VEL
LIN {X 0,Y 172.345,Z 432.392,A -85,B 0,C 180,E1 -23126.497,E2 -23126.497} C_VEL
LIN {X 0,Y 172.286,Z 439.337,A -85,B 0,C 180,E1 -23128.835,E2 -23128.835} C_VEL
LIN {X 0,Y 172.121,Z 445.031,A -85,B 0,C 180,E1 -23131.174,E2 -23131.174} C_VEL
LIN {X 0,Y 171.583,Z 449.635,A -85,B 0,C 180,E1 -23133.526,E2 -23133.526} C_VEL
LIN {X 0,Y 171.1,Z 453.501,A -85,B 0,C 180,E1 -23135.898,E2 -23135.898} C_VEL
LIN {X 0,Y 170.985,Z 458.029,A -85,B 0,C 180,E1 -23139.467,E2 -23139.467} C_VEL
LIN {X 0,Y 171.32,Z 460.502,A -85,B 0,C 180,E1 -23141.84,E2 -23141.84} C_VEL
LIN {X 0,Y 172.129,Z 462.466,A -85,B 0,C 180,E1 -23144.184,E2 -23144.184} C_VEL
LIN {X 0,Y 173.954,Z 464.502,A -85,B 0,C 180,E1 -23147.347,E2 -23147.347} C_VEL
LIN {X 0,Y 174.734,Z 465.343,A -85,B 0,C 180,E1 -23149.255,E2 -23149.255} C_VEL
LIN {X 0,Y 174.855,Z 465.905,A -85,B 0,C 180,E1 -23152.502,E2 -23152.502} C_VEL
LIN {X 0,Y 175.777,Z 465.945,A -85,B 0,C 180,E1 -23155.718,E2 -23155.718} C_VEL
LIN {X 0,Y 177.753,Z 465.801,A -85,B 0,C 180,E1 -23157.513,E2 -23157.513} C_VEL
LIN {X 0,Y 182.336,Z 465.225,A -85,B 0,C 180,E1 -23160.075,E2 -23160.075} C_VEL
LIN {X 0,Y 190.38,Z 462.74,A -85,B 0,C 180,E1 -23163.627,E2 -23163.627} C_VEL
LIN {X 0,Y 197.137,Z 459.771,A -85,B 0,C 180,E1 -23166.035,E2 -23166.035} C_VEL
LIN {X 0,Y 204.415,Z 455.667,A -85,B 0,C 180,E1 -23168.236,E2 -23168.236} C_VEL
LIN {X 0,Y 213.033,Z 449.814,A -85,B 0,C 180,E1 -23170.42,E2 -23170.42} C_VEL
LIN {X 0,Y 221.902,Z 442.298,A -85,B 0,C 180,E1 -23172.304,E2 -23172.304} C_VEL
LIN {X 0,Y 229.254,Z 435.003,A -85,B 0,C 180,E1 -23173.614,E2 -23173.614} C_VEL
LIN {X 0,Y 236.871,Z 426.089,A -85,B 0,C 180,E1 -23174.806,E2 -23174.806} C_VEL
LIN {X 0,Y 240.507,Z 421.105,A -85,B 0,C 180,E1 -23175.32,E2 -23175.32} C_VEL
LIN {X 0,Y 241.337,Z 419.907,A -85,B 0,C 180,E1 -23175.652,E2 -23175.652} C_VEL
LIN {X 0,Y 235.458,Z 427.518,A -85,B 0,C 180,E1 -23176.637,E2 -23176.637} C_VEL
LIN {X 0,Y 229.76,Z 433.832,A -85,B 0,C 180,E1 -23177.696,E2 -23177.696} C_VEL
LIN {X 0,Y 221.44,Z 441.712,A -85,B 0,C 180,E1 -23179.402,E2 -23179.402} C_VEL
LIN {X 0,Y 213.427,Z 447.839,A -85,B 0,C 180,E1 -23181.26,E2 -23181.26} C_VEL
LIN {X 0,Y 205.838,Z 452.521,A -85,B 0,C 180,E1 -23183.298,E2 -23183.298} C_VEL
LIN {X 0,Y 198.77,Z 456.005,A -85,B 0,C 180,E1 -23185.538,E2 -23185.538} C_VEL
LIN {X 0,Y 194.278,Z 457.706,A -85,B 0,C 180,E1 -23187.127,E2 -23187.127} C_VEL
LIN {X 0,Y 190.063,Z 458.995,A -85,B 0,C 180,E1 -23188.813,E2 -23188.813} C_VEL
LIN {X 0,Y 186.063,Z 459.739,A -85,B 0,C 180,E1 -23190.581,E2 -23190.581} C_VEL
LIN {X 0,Y 178.867,Z 459.995,A -85,B 0,C 180,E1 -23194.381,E2 -23194.381} C_VEL
LIN {X 0,Y 175.761,Z 459.471,A -85,B 0,C 180,E1 -23196.419,E2 -23196.419} C_VEL
LIN {X 0,Y 170.428,Z 457.073,A -85,B 0,C 180,E1 -23200.726,E2 -23200.726} C_VEL
LIN {X 0,Y 167.552,Z 454.165,A -85,B 0,C 180,E1 -23204.167,E2 -23204.167} C_VEL
LIN {X 0,Y 165.314,Z 450.186,A -85,B 0,C 180,E1 -23207.715,E2 -23207.715} C_VEL
LIN {X 0,Y 164.141,Z 445.174,A -85,B 0,C 180,E1 -23211.369,E2 -23211.369} C_VEL
LIN {X 0,Y 163.735,Z 438.839,A -85,B 0,C 180,E1 -23215.063,E2 -23215.063} C_VEL
LIN {X 0,Y 163.789,Z 430.762,A -85,B 0,C 180,E1 -23218.758,E2 -23218.758} C_VEL
LIN {X 0,Y 164.11,Z 424.23,A -85,B 0,C 180,E1 -23221.215,E2 -23221.215} C_VEL
LIN {X 0,Y 164.435,Z 415.075,A -85,B 0,C 180,E1 -23223.97,E2 -23223.97} C_VEL
LIN {X 0,Y 164.805,Z 405.033,A -85,B 0,C 180,E1 -23226.415,E2 -23226.415} C_VEL
LIN {X 0,Y 165.25,Z 393.594,A -85,B 0,C 180,E1 -23228.548,E2 -23228.548} C_VEL
LIN {X 0,Y 165.624,Z 383.162,A -85,B 0,C 180,E1 -23230.059,E2 -23230.059} C_VEL
LIN {X 0,Y 165.982,Z 369.823,A -85,B 0,C 180,E1 -23231.461,E2 -23231.461} C_VEL
LIN {X 0,Y 166.557,Z 321.277,A -85,B 0,C 180,E1 -23235.552,E2 -23235.552} C_VEL
LIN {X 0,Y 164.747,Z 304.941,A -85,B 0,C 180,E1 -23236.801,E2 -23236.801} C_VEL
LIN {X 0,Y 164.367,Z 304.818,A -85,B 0,C 180,E1 -23242.618,E2 -23242.618} C_VEL
LIN {X 0,Y 164.36,Z 304.824,A -85,B 0,C 180,E1 -23246.102,E2 -23246.102} C_VEL
LIN {X 0,Y 164.339,Z 304.819,A -85,B 0,C 180,E1 -23251.2,E2 -23251.2} C_VEL
LIN {X 0,Y 164.262,Z 304.836,A -85,B 0,C 180,E1 -23256.78,E2 -23256.78} C_VEL
LIN {X 0,Y 164.266,Z 304.831,A -85,B 0,C 180,E1 -23259.905,E2 -23259.905} C_VEL
LIN {X 0,Y 164.258,Z 304.835,A -85,B 0,C 180,E1 -23263.329,E2 -23263.329} C_VEL
LIN {X 0,Y 164.236,Z 304.839,A -85,B 0,C 180,E1 -23266.785,E2 -23266.785} C_VEL
LIN {X 0,Y 164.262,Z 304.83,A -85,B 0,C 180,E1 -23270.343,E2 -23270.343} C_VEL
LIN {X 0,Y 164.296,Z 304.831,A -85,B 0,C 180,E1 -23274.34,E2 -23274.34} C_VEL
LIN {X 0,Y 164.337,Z 304.822,A -85,B 0,C 180,E1 -23279.119,E2 -23279.119} C_VEL
LIN {X 0,Y 164.369,Z 304.821,A -85,B 0,C 180,E1 -23284.682,E2 -23284.682} C_VEL
LIN {X 0,Y 164.447,Z 304.812,A -85,B 0,C 180,E1 -23290.043,E2 -23290.043} C_VEL
LIN {X 0,Y 164.461,Z 304.809,A -85,B 0,C 180,E1 -23295.139,E2 -23295.139} C_VEL
LIN {X 0,Y 164.746,Z 304.776,A -85,B 0,C 180,E1 -23300.171,E2 -23300.171} C_VEL
LIN {X 0,Y 164.794,Z 304.768,A -85,B 0,C 180,E1 -23302.645,E2 -23302.645} C_VEL
LIN {X 0,Y 165.018,Z 304.739,A -85,B 0,C 180,E1 -23307.555,E2 -23307.555} C_VEL
LIN {X 0,Y 165.255,Z 304.714,A -85,B 0,C 180,E1 -23309.996,E2 -23309.996} C_VEL
LIN {X 0,Y 164.729,Z 304.772,A -85,B 0,C 180,E1 -23314.891,E2 -23314.891} C_VEL
LIN {X 0,Y 164.791,Z 304.768,A -85,B 0,C 180,E1 -23317.347,E2 -23317.347} C_VEL
LIN {X 0,Y 164.7,Z 304.779,A -85,B 0,C 180,E1 -23321.135,E2 -23321.135} C_VEL
LIN {X 0,Y 164.432,Z 304.814,A -85,B 0,C 180,E1 -23327.404,E2 -23327.404} C_VEL
LIN {X 0,Y 164.427,Z 304.814,A -85,B 0,C 180,E1 -23329.99,E2 -23329.99} C_VEL
LIN {X 0,Y 164.341,Z 304.825,A -85,B 0,C 180,E1 -23336.13,E2 -23336.13} C_VEL
LIN {X 0,Y 164.332,Z 304.822,A -85,B 0,C 180,E1 -23341.231,E2 -23341.231} C_VEL
LIN {X 0,Y 164.309,Z 304.831,A -85,B 0,C 180,E1 -23346.78,E2 -23346.78} C_VEL
LIN {X 0,Y 164.334,Z 304.821,A -85,B 0,C 180,E1 -23349.898,E2 -23349.898} C_VEL
LIN {X 0,Y 164.351,Z 304.826,A -85,B 0,C 180,E1 -23353.389,E2 -23353.389} C_VEL
LIN {X 0,Y 164.353,Z 304.824,A -85,B 0,C 180,E1 -23356.848,E2 -23356.848} C_VEL
LIN {X 0,Y 164.336,Z 304.822,A -85,B 0,C 180,E1 -23360.328,E2 -23360.328} C_VEL
LIN {X 0,Y 164.31,Z 304.829,A -85,B 0,C 180,E1 -23364.351,E2 -23364.351} C_VEL
LIN {X 0,Y 164.356,Z 304.818,A -85,B 0,C 180,E1 -23369.144,E2 -23369.144} C_VEL
LIN {X 0,Y 164.376,Z 304.82,A -85,B 0,C 180,E1 -23374.703,E2 -23374.703} C_VEL
LIN {X 0,Y 164.413,Z 304.817,A -85,B 0,C 180,E1 -23380.106,E2 -23380.106} C_VEL
LIN {X 0,Y 164.463,Z 304.807,A -85,B 0,C 180,E1 -23385.157,E2 -23385.157} C_VEL
LIN {X 0,Y 164.746,Z 304.777,A -85,B 0,C 180,E1 -23390.188,E2 -23390.188} C_VEL
LIN {X 0,Y 164.806,Z 304.767,A -85,B 0,C 180,E1 -23392.663,E2 -23392.663} C_VEL
LIN {X 0,Y 165.26,Z 304.711,A -85,B 0,C 180,E1 -23400.012,E2 -23400.012} C_VEL
LIN {X 0,Y 164.81,Z 304.767,A -85,B 0,C 180,E1 -23407.362,E2 -23407.362} C_VEL
LIN {X 0,Y 164.694,Z 304.78,A -85,B 0,C 180,E1 -23411.069,E2 -23411.069} C_VEL
LIN {X 0,Y 164.423,Z 304.816,A -85,B 0,C 180,E1 -23417.422,E2 -23417.422} C_VEL
LIN {X 0,Y 164.416,Z 304.814,A -85,B 0,C 180,E1 -23420.008,E2 -23420.008} C_VEL
LIN {X 0,Y 164.339,Z 304.825,A -85,B 0,C 180,E1 -23426.106,E2 -23426.106} C_VEL
LIN {X 0,Y 164.356,Z 304.82,A -85,B 0,C 180,E1 -23431.226,E2 -23431.226} C_VEL
LIN {X 0,Y 164.285,Z 304.832,A -85,B 0,C 180,E1 -23436.805,E2 -23436.805} C_VEL
LIN {X 0,Y 164.293,Z 304.826,A -85,B 0,C 180,E1 -23439.929,E2 -23439.929} C_VEL
LIN {X 0,Y 164.29,Z 304.831,A -85,B 0,C 180,E1 -23443.352,E2 -23443.352} C_VEL
LIN {X 0,Y 164.27,Z 304.833,A -85,B 0,C 180,E1 -23446.808,E2 -23446.808} C_VEL
LIN {X 0,Y 164.301,Z 304.828,A -85,B 0,C 180,E1 -23450.365,E2 -23450.365} C_VEL
LIN {X 0,Y 164.34,Z 304.824,A -85,B 0,C 180,E1 -23456.23,E2 -23456.23} C_VEL
LIN {X 0,Y 164.537,Z 304.802,A -85,B 0,C 180,E1 -23461.98,E2 -23461.98} C_VEL
LIN {X 0,Y 164.856,Z 304.763,A -85,B 0,C 180,E1 -23464.771,E2 -23464.771} C_VEL
LIN {X 0,Y 164.842,Z 304.764,A -85,B 0,C 180,E1 -23467.441,E2 -23467.441} C_VEL
LIN {X 0,Y 164.437,Z 304.886,A -85,B 0,C 180,E1 -23468.867,E2 -23468.867} C_VEL
LIN {X 0,Y 163.921,Z 310.766,A -85,B 0,C 180,E1 -23472.62,E2 -23472.62} C_VEL
LIN {X 0,Y 164.656,Z 332.728,A -85,B 0,C 180,E1 -23474.414,E2 -23474.414} C_VEL
LIN {X 0,Y 166.507,Z 353.835,A -85,B 0,C 180,E1 -23476.059,E2 -23476.059} C_VEL
LIN {X 0,Y 166.24,Z 390.286,A -85,B 0,C 180,E1 -23479.269,E2 -23479.269} C_VEL
LIN {X 0,Y 166.005,Z 402.596,A -85,B 0,C 180,E1 -23480.869,E2 -23480.869} C_VEL
LIN {X 0,Y 165.823,Z 412.939,A -85,B 0,C 180,E1 -23482.699,E2 -23482.699} C_VEL
LIN {X 0,Y 165.672,Z 423.758,A -85,B 0,C 180,E1 -23485.137,E2 -23485.137} C_VEL
LIN {X 0,Y 165.677,Z 432.188,A -85,B 0,C 180,E1 -23487.573,E2 -23487.573} C_VEL
LIN {X 0,Y 165.634,Z 439.056,A -85,B 0,C 180,E1 -23490.004,E2 -23490.004} C_VEL
LIN {X 0,Y 165.32,Z 444.619,A -85,B 0,C 180,E1 -23492.441,E2 -23492.441} C_VEL
LIN {X 0,Y 164.744,Z 449.052,A -85,B 0,C 180,E1 -23494.899,E2 -23494.899} C_VEL
LIN {X 0,Y 164.352,Z 452.805,A -85,B 0,C 180,E1 -23497.375,E2 -23497.375} C_VEL
LIN {X 0,Y 164.378,Z 457.255,A -85,B 0,C 180,E1 -23500.972,E2 -23500.972} C_VEL
LIN {X 0,Y 165.435,Z 460.858,A -85,B 0,C 180,E1 -23504.771,E2 -23504.771} C_VEL
LIN {X 0,Y 167.247,Z 463.162,A -85,B 0,C 180,E1 -23507.964,E2 -23507.964} C_VEL
LIN {X 0,Y 170.415,Z 465.089,A -85,B 0,C 180,E1 -23511.791,E2 -23511.791} C_VEL
LIN {X 0,Y 172.834,Z 465.739,A -85,B 0,C 180,E1 -23513.997,E2 -23513.997} C_VEL
LIN {X 0,Y 177.753,Z 465.801,A -85,B 0,C 180,E1 -23517.513,E2 -23517.513} C_VEL
LIN {X 0,Y 180.025,Z 465.588,A -85,B 0,C 180,E1 -23519.264,E2 -23519.264} C_VEL
LIN {X 0,Y 182.715,Z 464.764,A -85,B 0,C 180,E1 -23522.275,E2 -23522.275} C_VEL
LIN {X 0,Y 185.237,Z 463.572,A -85,B 0,C 180,E1 -23524.574,E2 -23524.574} C_VEL
LIN {X 0,Y 188.062,Z 462.299,A -85,B 0,C 180,E1 -23526.103,E2 -23526.103} C_VEL
LIN {X 0,Y 189.257,Z 461.796,A -85,B 0,C 180,E1 -23526.547,E2 -23526.547} C_VEL
LIN {X 0,Y 196.394,Z 458.73,A -85,B 0,C 180,E1 -23528.777,E2 -23528.777} C_VEL
LIN {X 0,Y 205.031,Z 454.045,A -85,B 0,C 180,E1 -23531.041,E2 -23531.041} C_VEL
LIN {X 0,Y 213.937,Z 447.992,A -85,B 0,C 180,E1 -23532.977,E2 -23532.977} C_VEL
LIN {X 0,Y 221.305,Z 442.012,A -85,B 0,C 180,E1 -23534.323,E2 -23534.323} C_VEL
LIN {X 0,Y 228.708,Z 434.911,A -85,B 0,C 180,E1 -23535.497,E2 -23535.497} C_VEL
LIN {X 0,Y 227.865,Z 435.721,A -85,B 0,C 180,E1 -23536.046,E2 -23536.046} C_VEL
LIN {X 0,Y 219.208,Z 443.266,A -85,B 0,C 180,E1 -23537.67,E2 -23537.67} C_VEL
LIN {X 0,Y 210.86,Z 449.074,A -85,B 0,C 180,E1 -23539.453,E2 -23539.453} C_VEL
LIN {X 0,Y 202.92,Z 453.602,A -85,B 0,C 180,E1 -23541.424,E2 -23541.424} C_VEL
LIN {X 0,Y 197.871,Z 455.902,A -85,B 0,C 180,E1 -23542.847,E2 -23542.847} C_VEL
LIN {X 0,Y 193.083,Z 457.767,A -85,B 0,C 180,E1 -23544.371,E2 -23544.371} C_VEL
LIN {X 0,Y 188.434,Z 459.123,A -85,B 0,C 180,E1 -23545.971,E2 -23545.971} C_VEL
LIN {X 0,Y 179.95,Z 460.445,A -85,B 0,C 180,E1 -23549.477,E2 -23549.477} C_VEL
LIN {X 0,Y 176.11,Z 460.526,A -85,B 0,C 180,E1 -23551.376,E2 -23551.376} C_VEL
LIN {X 0,Y 169.291,Z 459.248,A -85,B 0,C 180,E1 -23555.46,E2 -23555.46} C_VEL
LIN {X 0,Y 166.348,Z 458.063,A -85,B 0,C 180,E1 -23557.64,E2 -23557.64} C_VEL
LIN {X 0,Y 162.752,Z 455.389,A -85,B 0,C 180,E1 -23561.091,E2 -23561.091} C_VEL
LIN {X 0,Y 159.936,Z 451.734,A -85,B 0,C 180,E1 -23564.701,E2 -23564.701} C_VEL
LIN {X 0,Y 158.161,Z 447.292,A -85,B 0,C 180,E1 -23568.207,E2 -23568.207} C_VEL
LIN {X 0,Y 157.218,Z 441.077,A -85,B 0,C 180,E1 -23572.281,E2 -23572.281} C_VEL
LIN {X 0,Y 156.995,Z 435.048,A -85,B 0,C 180,E1 -23575.494,E2 -23575.494} C_VEL
LIN {X 0,Y 157.174,Z 427.731,A -85,B 0,C 180,E1 -23578.706,E2 -23578.706} C_VEL
LIN {X 0,Y 157.45,Z 419.695,A -85,B 0,C 180,E1 -23581.586,E2 -23581.586} C_VEL
LIN {X 0,Y 157.772,Z 410.824,A -85,B 0,C 180,E1 -23584.138,E2 -23584.138} C_VEL
LIN {X 0,Y 158.106,Z 401.022,A -85,B 0,C 180,E1 -23586.367,E2 -23586.367} C_VEL
LIN {X 0,Y 158.515,Z 389.593,A -85,B 0,C 180,E1 -23588.432,E2 -23588.432} C_VEL
LIN {X 0,Y 158.961,Z 377.549,A -85,B 0,C 180,E1 -23590.012,E2 -23590.012} C_VEL
LIN {X 0,Y 159.198,Z 356.485,A -85,B 0,C 180,E1 -23592.01,E2 -23592.01} C_VEL
LIN {X 0,Y 159.494,Z 321.057,A -85,B 0,C 180,E1 -23595.183,E2 -23595.183} C_VEL
LIN {X 0,Y 157.773,Z 305.728,A -85,B 0,C 180,E1 -23596.4,E2 -23596.4} C_VEL
LIN {X 0,Y 157.294,Z 305.699,A -85,B 0,C 180,E1 -23603.696,E2 -23603.696} C_VEL
LIN {X 0,Y 157.301,Z 305.703,A -85,B 0,C 180,E1 -23606.666,E2 -23606.666} C_VEL
LIN {X 0,Y 157.25,Z 305.705,A -85,B 0,C 180,E1 -23612.416,E2 -23612.416} C_VEL
LIN {X 0,Y 157.241,Z 305.712,A -85,B 0,C 180,E1 -23616.43,E2 -23616.43} C_VEL
LIN {X 0,Y 157.168,Z 305.715,A -85,B 0,C 180,E1 -23622.104,E2 -23622.104} C_VEL
LIN {X 0,Y 157.165,Z 305.716,A -85,B 0,C 180,E1 -23627.869,E2 -23627.869} C_VEL
LIN {X 0,Y 157.229,Z 305.712,A -85,B 0,C 180,E1 -23633.544,E2 -23633.544} C_VEL
LIN {X 0,Y 157.25,Z 305.703,A -85,B 0,C 180,E1 -23638.092,E2 -23638.092} C_VEL
LIN {X 0,Y 157.276,Z 305.707,A -85,B 0,C 180,E1 -23643.453,E2 -23643.453} C_VEL
LIN {X 0,Y 157.355,Z 305.696,A -85,B 0,C 180,E1 -23649.661,E2 -23649.661} C_VEL
LIN {X 0,Y 157.398,Z 305.688,A -85,B 0,C 180,E1 -23654.456,E2 -23654.456} C_VEL
LIN {X 0,Y 157.677,Z 305.657,A -85,B 0,C 180,E1 -23659.726,E2 -23659.726} C_VEL
LIN {X 0,Y 157.733,Z 305.648,A -85,B 0,C 180,E1 -23662.314,E2 -23662.314} C_VEL
LIN {X 0,Y 157.966,Z 305.617,A -85,B 0,C 180,E1 -23667.446,E2 -23667.446} C_VEL
LIN {X 0,Y 158.217,Z 305.591,A -85,B 0,C 180,E1 -23669.996,E2 -23669.996} C_VEL
LIN {X 0,Y 157.677,Z 305.65,A -85,B 0,C 180,E1 -23675.11,E2 -23675.11} C_VEL
LIN {X 0,Y 157.729,Z 305.648,A -85,B 0,C 180,E1 -23677.677,E2 -23677.677} C_VEL
LIN {X 0,Y 157.629,Z 305.659,A -85,B 0,C 180,E1 -23681.302,E2 -23681.302} C_VEL
LIN {X 0,Y 157.361,Z 305.696,A -85,B 0,C 180,E1 -23688.213,E2 -23688.213} C_VEL
LIN {X 0,Y 157.257,Z 305.704,A -85,B 0,C 180,E1 -23693.712,E2 -23693.712} C_VEL
LIN {X 0,Y 157.265,Z 305.709,A -85,B 0,C 180,E1 -23696.684,E2 -23696.684} C_VEL
LIN {X 0,Y 157.235,Z 305.706,A -85,B 0,C 180,E1 -23702.431,E2 -23702.431} C_VEL
LIN {X 0,Y 157.283,Z 305.705,A -85,B 0,C 180,E1 -23706.483,E2 -23706.483} C_VEL
LIN {X 0,Y 157.255,Z 305.705,A -85,B 0,C 180,E1 -23712.089,E2 -23712.089} C_VEL
LIN {X 0,Y 157.272,Z 305.706,A -85,B 0,C 180,E1 -23715.635,E2 -23715.635} C_VEL
LIN {X 0,Y 157.252,Z 305.706,A -85,B 0,C 180,E1 -23721.286,E2 -23721.286} C_VEL
LIN {X 0,Y 157.257,Z 305.708,A -85,B 0,C 180,E1 -23724.498,E2 -23724.498} C_VEL
LIN {X 0,Y 157.26,Z 305.701,A -85,B 0,C 180,E1 -23728.106,E2 -23728.106} C_VEL
LIN {X 0,Y 157.284,Z 305.706,A -85,B 0,C 180,E1 -23733.475,E2 -23733.475} C_VEL
LIN {X 0,Y 157.351,Z 305.694,A -85,B 0,C 180,E1 -23739.696,E2 -23739.696} C_VEL
LIN {X 0,Y 157.398,Z 305.688,A -85,B 0,C 180,E1 -23744.474,E2 -23744.474} C_VEL
LIN {X 0,Y 157.668,Z 305.656,A -85,B 0,C 180,E1 -23749.743,E2 -23749.743} C_VEL
LIN {X 0,Y 157.743,Z 305.648,A -85,B 0,C 180,E1 -23752.332,E2 -23752.332} C_VEL
LIN {X 0,Y 158.223,Z 305.588,A -85,B 0,C 180,E1 -23760.013,E2 -23760.013} C_VEL
LIN {X 0,Y 157.748,Z 305.646,A -85,B 0,C 180,E1 -23767.693,E2 -23767.693} C_VEL
LIN {X 0,Y 157.623,Z 305.66,A -85,B 0,C 180,E1 -23771.235,E2 -23771.235} C_VEL
LIN {X 0,Y 157.4,Z 305.689,A -85,B 0,C 180,E1 -23775.552,E2 -23775.552} C_VEL
LIN {X 0,Y 157.3,Z 305.7,A -85,B 0,C 180,E1 -23780.955,E2 -23780.955} C_VEL
LIN {X 0,Y 157.268,Z 305.707,A -85,B 0,C 180,E1 -23786.661,E2 -23786.661} C_VEL
LIN {X 0,Y 157.268,Z 305.702,A -85,B 0,C 180,E1 -23792.442,E2 -23792.442} C_VEL
LIN {X 0,Y 157.264,Z 305.707,A -85,B 0,C 180,E1 -23796.456,E2 -23796.456} C_VEL
LIN {X 0,Y 157.198,Z 305.714,A -85,B 0,C 180,E1 -23802.129,E2 -23802.129} C_VEL
LIN {X 0,Y 157.2,Z 305.712,A -85,B 0,C 180,E1 -23807.892,E2 -23807.892} C_VEL
LIN {X 0,Y 157.272,Z 305.706,A -85,B 0,C 180,E1 -23813.566,E2 -23813.566} C_VEL
LIN {X 0,Y 157.309,Z 305.697,A -85,B 0,C 180,E1 -23818.106,E2 -23818.106} C_VEL
LIN {X 0,Y 157.668,Z 305.657,A -85,B 0,C 180,E1 -23823.534,E2 -23823.534} C_VEL
LIN {X 0,Y 157.779,Z 305.645,A -85,B 0,C 180,E1 -23826.371,E2 -23826.371} C_VEL
LIN {X 0,Y 157.131,Z 305.882,A -85,B 0,C 180,E1 -23829.883,E2 -23829.883} C_VEL
LIN {X 0,Y 156.893,Z 310.739,A -85,B 0,C 180,E1 -23832.993,E2 -23832.993} C_VEL
LIN {X 0,Y 157.681,Z 332.831,A -85,B 0,C 180,E1 -23834.865,E2 -23834.865} C_VEL
LIN {X 0,Y 159.582,Z 353.397,A -85,B 0,C 180,E1 -23836.541,E2 -23836.541} C_VEL
LIN {X 0,Y 159.458,Z 389.511,A -85,B 0,C 180,E1 -23839.93,E2 -23839.93} C_VEL
LIN {X 0,Y 159.288,Z 400.868,A -85,B 0,C 180,E1 -23841.441,E2 -23841.441} C_VEL
LIN {X 0,Y 159.13,Z 411.41,A -85,B 0,C 180,E1 -23843.347,E2 -23843.347} C_VEL
LIN {X 0,Y 159.054,Z 421.186,A -85,B 0,C 180,E1 -23845.569,E2 -23845.569} C_VEL
LIN {X 0,Y 159.047,Z 430.125,A -85,B 0,C 180,E1 -23848.105,E2 -23848.105} C_VEL
LIN {X 0,Y 159.026,Z 437.171,A -85,B 0,C 180,E1 -23850.637,E2 -23850.637} C_VEL
LIN {X 0,Y 158.679,Z 442.777,A -85,B 0,C 180,E1 -23853.178,E2 -23853.178} C_VEL
LIN {X 0,Y 157.955,Z 448.329,A -85,B 0,C 180,E1 -23856.391,E2 -23856.391} C_VEL
LIN {X 0,Y 157.695,Z 453.639,A -85,B 0,C 180,E1 -23860.273,E2 -23860.273} C_VEL
LIN {X 0,Y 158.371,Z 457.812,A -85,B 0,C 180,E1 -23864.131,E2 -23864.131} C_VEL
LIN {X 0,Y 160.129,Z 461.084,A -85,B 0,C 180,E1 -23867.896,E2 -23867.896} C_VEL
LIN {X 0,Y 161.827,Z 462.777,A -85,B 0,C 180,E1 -23870.335,E2 -23870.335} C_VEL
LIN {X 0,Y 166.441,Z 464.85,A -85,B 0,C 180,E1 -23874.981,E2 -23874.981} C_VEL
LIN {X 0,Y 169.251,Z 465.394,A -85,B 0,C 180,E1 -23877.183,E2 -23877.183} C_VEL
LIN {X 0,Y 172.587,Z 465.473,A -85,B 0,C 180,E1 -23879.257,E2 -23879.257} C_VEL
LIN {X 0,Y 180.245,Z 464.543,A -85,B 0,C 180,E1 -23883.089,E2 -23883.089} C_VEL
LIN {X 0,Y 184.528,Z 463.426,A -85,B 0,C 180,E1 -23884.845,E2 -23884.845} C_VEL
LIN {X 0,Y 189.257,Z 461.796,A -85,B 0,C 180,E1 -23886.547,E2 -23886.547} C_VEL
LIN {X 0,Y 192.669,Z 460.378,A -85,B 0,C 180,E1 -23887.927,E2 -23887.927} C_VEL
LIN {X 0,Y 201.171,Z 455.511,A -85,B 0,C 180,E1 -23892.268,E2 -23892.268} C_VEL
LIN {X 0,Y 204.747,Z 453.344,A -85,B 0,C 180,E1 -23893.422,E2 -23893.422} C_VEL
LIN {X 0,Y 206.117,Z 452.481,A -85,B 0,C 180,E1 -23893.731,E2 -23893.731} C_VEL
LIN {X 0,Y 214.861,Z 446.607,A -85,B 0,C 180,E1 -23895.355,E2 -23895.355} C_VEL
LIN {X 0,Y 216.377,Z 445.444,A -85,B 0,C 180,E1 -23895.612,E2 -23895.612} C_VEL
LIN {X 0,Y 214.281,Z 446.892,A -85,B 0,C 180,E1 -23896.458,E2 -23896.458} C_VEL
LIN {X 0,Y 205.742,Z 452.06,A -85,B 0,C 180,E1 -23898.223,E2 -23898.223} C_VEL
LIN {X 0,Y 197.552,Z 455.882,A -85,B 0,C 180,E1 -23900.171,E2 -23900.171} C_VEL
LIN {X 0,Y 192.395,Z 457.839,A -85,B 0,C 180,E1 -23901.601,E2 -23901.601} C_VEL
LIN {X 0,Y 182.652,Z 460.219,A -85,B 0,C 180,E1 -23904.738,E2 -23904.738} C_VEL
LIN {X 0,Y 178.137,Z 460.857,A -85,B 0,C 180,E1 -23906.461,E2 -23906.461} C_VEL
LIN {X 0,Y 170.799,Z 460.764,A -85,B 0,C 180,E1 -23909.787,E2 -23909.787} C_VEL
LIN {X 0,Y 166.195,Z 460.003,A -85,B 0,C 180,E1 -23912.267,E2 -23912.267} C_VEL
LIN {X 0,Y 162.886,Z 458.881,A -85,B 0,C 180,E1 -23914.427,E2 -23914.427} C_VEL
LIN {X 0,Y 157.21,Z 455.396,A -85,B 0,C 180,E1 -23919.032,E2 -23919.032} C_VEL
LIN {X 0,Y 154.168,Z 451.648,A -85,B 0,C 180,E1 -23922.751,E2 -23922.751} C_VEL
LIN {X 0,Y 151.879,Z 446.868,A -85,B 0,C 180,E1 -23926.609,E2 -23926.609} C_VEL
LIN {X 0,Y 150.726,Z 440.93,A -85,B 0,C 180,E1 -23930.594,E2 -23930.594} C_VEL
LIN {X 0,Y 150.389,Z 433.683,A -85,B 0,C 180,E1 -23934.624,E2 -23934.624} C_VEL
LIN {X 0,Y 150.511,Z 426.146,A -85,B 0,C 180,E1 -23937.98,E2 -23937.98} C_VEL
LIN {X 0,Y 150.815,Z 418.742,A -85,B 0,C 180,E1 -23940.654,E2 -23940.654} C_VEL
LIN {X 0,Y 151.124,Z 409.684,A -85,B 0,C 180,E1 -23943.319,E2 -23943.319} C_VEL
LIN {X 0,Y 151.379,Z 399.849,A -85,B 0,C 180,E1 -23945.648,E2 -23945.648} C_VEL
LIN {X 0,Y 151.755,Z 388.234,A -85,B 0,C 180,E1 -23947.805,E2 -23947.805} C_VEL
LIN {X 0,Y 152.135,Z 377.216,A -85,B 0,C 180,E1 -23949.291,E2 -23949.291} C_VEL
LIN {X 0,Y 152.354,Z 350.958,A -85,B 0,C 180,E1 -23951.882,E2 -23951.882} C_VEL
LIN {X 0,Y 152.428,Z 320.468,A -85,B 0,C 180,E1 -23954.732,E2 -23954.732} C_VEL
LIN {X 0,Y 150.844,Z 306.508,A -85,B 0,C 180,E1 -23955.94,E2 -23955.94} C_VEL
LIN {X 0,Y 150.259,Z 306.575,A -85,B 0,C 180,E1 -23961.958,E2 -23961.958} C_VEL
LIN {X 0,Y 150.201,Z 306.588,A -85,B 0,C 180,E1 -23967.882,E2 -23967.882} C_VEL
LIN {X 0,Y 150.191,Z 306.585,A -85,B 0,C 180,E1 -23972.611,E2 -23972.611} C_VEL
LIN {X 0,Y 150.152,Z 306.592,A -85,B 0,C 180,E1 -23977.46,E2 -23977.46} C_VEL
LIN {X 0,Y 150.111,Z 306.594,A -85,B 0,C 180,E1 -23981.482,E2 -23981.482} C_VEL
LIN {X 0,Y 150.103,Z 306.599,A -85,B 0,C 180,E1 -23985.381,E2 -23985.381} C_VEL
LIN {X 0,Y 150.111,Z 306.593,A -85,B 0,C 180,E1 -23989.04,E2 -23989.04} C_VEL
LIN {X 0,Y 150.148,Z 306.593,A -85,B 0,C 180,E1 -23992.697,E2 -23992.697} C_VEL
LIN {X 0,Y 150.175,Z 306.585,A -85,B 0,C 180,E1 -23997.362,E2 -23997.362} C_VEL
LIN {X 0,Y 150.206,Z 306.586,A -85,B 0,C 180,E1 -24002.711,E2 -24002.711} C_VEL
LIN {X 0,Y 150.312,Z 306.57,A -85,B 0,C 180,E1 -24009.201,E2 -24009.201} C_VEL
LIN {X 0,Y 150.31,Z 306.573,A -85,B 0,C 180,E1 -24013.703,E2 -24013.703} C_VEL
LIN {X 0,Y 150.604,Z 306.535,A -85,B 0,C 180,E1 -24019.238,E2 -24019.238} C_VEL
LIN {X 0,Y 150.673,Z 306.529,A -85,B 0,C 180,E1 -24021.952,E2 -24021.952} C_VEL
LIN {X 0,Y 150.888,Z 306.498,A -85,B 0,C 180,E1 -24027.326,E2 -24027.326} C_VEL
LIN {X 0,Y 151.18,Z 306.467,A -85,B 0,C 180,E1 -24029.995,E2 -24029.995} C_VEL
LIN {X 0,Y 150.623,Z 306.529,A -85,B 0,C 180,E1 -24035.35,E2 -24035.35} C_VEL
LIN {X 0,Y 150.67,Z 306.529,A -85,B 0,C 180,E1 -24038.039,E2 -24038.039} C_VEL
LIN {X 0,Y 150.56,Z 306.54,A -85,B 0,C 180,E1 -24041.488,E2 -24041.488} C_VEL
LIN {X 0,Y 150.304,Z 306.574,A -85,B 0,C 180,E1 -24046.288,E2 -24046.288} C_VEL
LIN {X 0,Y 150.304,Z 306.571,A -85,B 0,C 180,E1 -24050.791,E2 -24050.791} C_VEL
LIN {X 0,Y 150.197,Z 306.588,A -85,B 0,C 180,E1 -24057.282,E2 -24057.282} C_VEL
LIN {X 0,Y 150.175,Z 306.585,A -85,B 0,C 180,E1 -24062.638,E2 -24062.638} C_VEL
LIN {X 0,Y 150.195,Z 306.587,A -85,B 0,C 180,E1 -24067.461,E2 -24067.461} C_VEL
LIN {X 0,Y 150.196,Z 306.585,A -85,B 0,C 180,E1 -24071.548,E2 -24071.548} C_VEL
LIN {X 0,Y 150.222,Z 306.585,A -85,B 0,C 180,E1 -24075.454,E2 -24075.454} C_VEL
LIN {X 0,Y 150.196,Z 306.583,A -85,B 0,C 180,E1 -24079.094,E2 -24079.094} C_VEL
LIN {X 0,Y 150.201,Z 306.586,A -85,B 0,C 180,E1 -24082.689,E2 -24082.689} C_VEL
LIN {X 0,Y 150.184,Z 306.586,A -85,B 0,C 180,E1 -24087.377,E2 -24087.377} C_VEL
LIN {X 0,Y 150.211,Z 306.585,A -85,B 0,C 180,E1 -24092.732,E2 -24092.732} C_VEL
LIN {X 0,Y 150.313,Z 306.57,A -85,B 0,C 180,E1 -24099.232,E2 -24099.232} C_VEL
LIN {X 0,Y 150.305,Z 306.575,A -85,B 0,C 180,E1 -24103.722,E2 -24103.722} C_VEL
LIN {X 0,Y 150.588,Z 306.537,A -85,B 0,C 180,E1 -24109.255,E2 -24109.255} C_VEL
LIN {X 0,Y 150.681,Z 306.528,A -85,B 0,C 180,E1 -24111.971,E2 -24111.971} C_VEL
LIN {X 0,Y 151.183,Z 306.465,A -85,B 0,C 180,E1 -24120.013,E2 -24120.013} C_VEL
LIN {X 0,Y 150.671,Z 306.528,A -85,B 0,C 180,E1 -24128.057,E2 -24128.057} C_VEL
LIN {X 0,Y 150.565,Z 306.539,A -85,B 0,C 180,E1 -24131.44,E2 -24131.44} C_VEL
LIN {X 0,Y 150.306,Z 306.572,A -85,B 0,C 180,E1 -24136.306,E2 -24136.306} C_VEL
LIN {X 0,Y 150.279,Z 306.576,A -85,B 0,C 180,E1 -24140.735,E2 -24140.735} C_VEL
LIN {X 0,Y 150.186,Z 306.591,A -85,B 0,C 180,E1 -24147.25,E2 -24147.25} C_VEL
LIN {X 0,Y 150.209,Z 306.581,A -85,B 0,C 180,E1 -24152.638,E2 -24152.638} C_VEL
LIN {X 0,Y 150.176,Z 306.591,A -85,B 0,C 180,E1 -24157.487,E2 -24157.487} C_VEL
LIN {X 0,Y 150.14,Z 306.59,A -85,B 0,C 180,E1 -24161.508,E2 -24161.508} C_VEL
LIN {X 0,Y 150.137,Z 306.596,A -85,B 0,C 180,E1 -24165.407,E2 -24165.407} C_VEL
LIN {X 0,Y 150.148,Z 306.588,A -85,B 0,C 180,E1 -24169.064,E2 -24169.064} C_VEL
LIN {X 0,Y 150.189,Z 306.588,A -85,B 0,C 180,E1 -24172.721,E2 -24172.721} C_VEL
LIN {X 0,Y 150.23,Z 306.58,A -85,B 0,C 180,E1 -24177.379,E2 -24177.379} C_VEL
LIN {X 0,Y 150.477,Z 306.553,A -85,B 0,C 180,E1 -24182.57,E2 -24182.57} C_VEL
LIN {X 0,Y 150.664,Z 306.53,A -85,B 0,C 180,E1 -24185.182,E2 -24185.182} C_VEL
LIN {X 0,Y 150.135,Z 306.597,A -85,B 0,C 180,E1 -24189.456,E2 -24189.456} C_VEL
LIN {X 0,Y 149.852,Z 306.753,A -85,B 0,C 180,E1 -24190.929,E2 -24190.929} C_VEL
LIN {X 0,Y 149.909,Z 310.361,A -85,B 0,C 180,E1 -24193.405,E2 -24193.405} C_VEL
LIN {X 0,Y 150.746,Z 332.536,A -85,B 0,C 180,E1 -24195.408,E2 -24195.408} C_VEL
LIN {X 0,Y 152.685,Z 353.531,A -85,B 0,C 180,E1 -24197.207,E2 -24197.207} C_VEL
LIN {X 0,Y 152.713,Z 388.527,A -85,B 0,C 180,E1 -24200.652,E2 -24200.652} C_VEL
LIN {X 0,Y 152.562,Z 401.016,A -85,B 0,C 180,E1 -24202.394,E2 -24202.394} C_VEL
LIN {X 0,Y 152.444,Z 411.419,A -85,B 0,C 180,E1 -24204.382,E2 -24204.382} C_VEL
LIN {X 0,Y 152.468,Z 419.743,A -85,B 0,C 180,E1 -24206.371,E2 -24206.371} C_VEL
LIN {X 0,Y 152.542,Z 429.698,A -85,B 0,C 180,E1 -24209.345,E2 -24209.345} C_VEL
LIN {X 0,Y 152.487,Z 436.589,A -85,B 0,C 180,E1 -24211.985,E2 -24211.985} C_VEL
LIN {X 0,Y 151.964,Z 442.054,A -85,B 0,C 180,E1 -24214.647,E2 -24214.647} C_VEL
LIN {X 0,Y 151.326,Z 447.516,A -85,B 0,C 180,E1 -24218.013,E2 -24218.013} C_VEL
LIN {X 0,Y 151.367,Z 453.542,A -85,B 0,C 180,E1 -24222.784,E2 -24222.784} C_VEL
LIN {X 0,Y 152.273,Z 456.998,A -85,B 0,C 180,E1 -24226.081,E2 -24226.081} C_VEL
LIN {X 0,Y 153.595,Z 459.328,A -85,B 0,C 180,E1 -24228.685,E2 -24228.685} C_VEL
LIN {X 0,Y 157.525,Z 462.705,A -85,B 0,C 180,E1 -24233.679,E2 -24233.679} C_VEL
LIN {X 0,Y 160.099,Z 463.868,A -85,B 0,C 180,E1 -24236.043,E2 -24236.043} C_VEL
LIN {X 0,Y 163.013,Z 464.548,A -85,B 0,C 180,E1 -24238.314,E2 -24238.314} C_VEL
LIN {X 0,Y 170.213,Z 465.03,A -85,B 0,C 180,E1 -24242.468,E2 -24242.468} C_VEL
LIN {X 0,Y 178.743,Z 463.838,A -85,B 0,C 180,E1 -24246.146,E2 -24246.146} C_VEL
LIN {X 0,Y 184.222,Z 462.435,A -85,B 0,C 180,E1 -24248.053,E2 -24248.053} C_VEL
LIN {X 0,Y 190.952,Z 460.127,A -85,B 0,C 180,E1 -24250.101,E2 -24250.101} C_VEL
LIN {X 0,Y 199.708,Z 456.064,A -85,B 0,C 180,E1 -24252.341,E2 -24252.341} C_VEL
LIN {X 0,Y 206.117,Z 452.481,A -85,B 0,C 180,E1 -24253.731,E2 -24253.731} C_VEL
LIN {X 0,Y 206.814,Z 452.016,A -85,B 0,C 180,E1 -24254.12,E2 -24254.12} C_VEL
LIN {X 0,Y 206.462,Z 452.022,A -85,B 0,C 180,E1 -24254.924,E2 -24254.924} C_VEL
LIN {X 0,Y 204.103,Z 453.072,A -85,B 0,C 180,E1 -24256.073,E2 -24256.073} C_VEL
LIN {X 0,Y 201.669,Z 454.152,A -85,B 0,C 180,E1 -24256.809,E2 -24256.809} C_VEL
LIN {X 0,Y 193.795,Z 457.329,A -85,B 0,C 180,E1 -24258.604,E2 -24258.604} C_VEL
LIN {X 0,Y 189.798,Z 458.662,A -85,B 0,C 180,E1 -24259.538,E2 -24259.538} C_VEL
LIN {X 0,Y 185.919,Z 459.605,A -85,B 0,C 180,E1 -24260.566,E2 -24260.566} C_VEL
LIN {X 0,Y 181.833,Z 460.517,A -85,B 0,C 180,E1 -24261.788,E2 -24261.788} C_VEL
LIN {X 0,Y 176.928,Z 461.207,A -85,B 0,C 180,E1 -24263.416,E2 -24263.416} C_VEL
LIN {X 0,Y 167.891,Z 461.218,A -85,B 0,C 180,E1 -24267.019,E2 -24267.019} C_VEL
LIN {X 0,Y 163.785,Z 460.677,A -85,B 0,C 180,E1 -24268.995,E2 -24268.995} C_VEL
LIN {X 0,Y 156.549,Z 458.223,A -85,B 0,C 180,E1 -24273.312,E2 -24273.312} C_VEL
LIN {X 0,Y 152.017,Z 455.323,A -85,B 0,C 180,E1 -24276.848,E2 -24276.848} C_VEL
LIN {X 0,Y 148.566,Z 451.544,A -85,B 0,C 180,E1 -24280.649,E2 -24280.649} C_VEL
LIN {X 0,Y 145.67,Z 446.023,A -85,B 0,C 180,E1 -24285.096,E2 -24285.096} C_VEL
LIN {X 0,Y 144.111,Z 438.51,A -85,B 0,C 180,E1 -24290.159,E2 -24290.159} C_VEL
LIN {X 0,Y 143.878,Z 432.025,A -85,B 0,C 180,E1 -24293.676,E2 -24293.676} C_VEL
LIN {X 0,Y 143.982,Z 424.199,A -85,B 0,C 180,E1 -24297.188,E2 -24297.188} C_VEL
LIN {X 0,Y 144.244,Z 417.731,A -85,B 0,C 180,E1 -24299.637,E2 -24299.637} C_VEL
LIN {X 0,Y 144.486,Z 408.521,A -85,B 0,C 180,E1 -24302.425,E2 -24302.425} C_VEL
LIN {X 0,Y 144.715,Z 398.477,A -85,B 0,C 180,E1 -24304.861,E2 -24304.861} C_VEL
LIN {X 0,Y 145.09,Z 387.354,A -85,B 0,C 180,E1 -24306.941,E2 -24306.941} C_VEL
LIN {X 0,Y 145.414,Z 376.305,A -85,B 0,C 180,E1 -24308.497,E2 -24308.497} C_VEL
LIN {X 0,Y 145.544,Z 345.418,A -85,B 0,C 180,E1 -24311.739,E2 -24311.739} C_VEL
LIN {X 0,Y 145.516,Z 320.97,A -85,B 0,C 180,E1 -24314.139,E2 -24314.139} C_VEL
LIN {X 0,Y 143.968,Z 307.364,A -85,B 0,C 180,E1 -24315.337,E2 -24315.337} C_VEL
LIN {X 0,Y 143.172,Z 307.457,A -85,B 0,C 180,E1 -24323.106,E2 -24323.106} C_VEL
LIN {X 0,Y 143.172,Z 307.463,A -85,B 0,C 180,E1 -24327.914,E2 -24327.914} C_VEL
LIN {X 0,Y 143.121,Z 307.466,A -85,B 0,C 180,E1 -24333.399,E2 -24333.399} C_VEL
LIN {X 0,Y 143.032,Z 307.475,A -85,B 0,C 180,E1 -24339.679,E2 -24339.679} C_VEL
LIN {X 0,Y 143.011,Z 307.482,A -85,B 0,C 180,E1 -24343.449,E2 -24343.449} C_VEL
LIN {X 0,Y 143.013,Z 307.479,A -85,B 0,C 180,E1 -24347.464,E2 -24347.464} C_VEL
LIN {X 0,Y 143.044,Z 307.477,A -85,B 0,C 180,E1 -24351.796,E2 -24351.796} C_VEL
LIN {X 0,Y 143.142,Z 307.461,A -85,B 0,C 180,E1 -24357.306,E2 -24357.306} C_VEL
LIN {X 0,Y 143.151,Z 307.465,A -85,B 0,C 180,E1 -24362.057,E2 -24362.057} C_VEL
LIN {X 0,Y 143.238,Z 307.45,A -85,B 0,C 180,E1 -24368.739,E2 -24368.739} C_VEL
LIN {X 0,Y 143.254,Z 307.452,A -85,B 0,C 180,E1 -24372.876,E2 -24372.876} C_VEL
LIN {X 0,Y 143.555,Z 307.413,A -85,B 0,C 180,E1 -24378.702,E2 -24378.702} C_VEL
LIN {X 0,Y 143.598,Z 307.411,A -85,B 0,C 180,E1 -24381.552,E2 -24381.552} C_VEL
LIN {X 0,Y 144.14,Z 307.344,A -85,B 0,C 180,E1 -24389.995,E2 -24389.995} C_VEL
LIN {X 0,Y 143.595,Z 307.411,A -85,B 0,C 180,E1 -24398.438,E2 -24398.438} C_VEL
LIN {X 0,Y 143.504,Z 307.419,A -85,B 0,C 180,E1 -24401.711,E2 -24401.711} C_VEL
LIN {X 0,Y 143.247,Z 307.453,A -85,B 0,C 180,E1 -24407.115,E2 -24407.115} C_VEL
LIN {X 0,Y 143.23,Z 307.451,A -85,B 0,C 180,E1 -24411.253,E2 -24411.253} C_VEL
LIN {X 0,Y 143.145,Z 307.466,A -85,B 0,C 180,E1 -24417.938,E2 -24417.938} C_VEL
LIN {X 0,Y 143.127,Z 307.467,A -85,B 0,C 180,E1 -24423.44,E2 -24423.44} C_VEL
LIN {X 0,Y 143.088,Z 307.467,A -85,B 0,C 180,E1 -24429.674,E2 -24429.674} C_VEL
LIN {X 0,Y 143.142,Z 307.467,A -85,B 0,C 180,E1 -24433.415,E2 -24433.415} C_VEL
LIN {X 0,Y 143.124,Z 307.466,A -85,B 0,C 180,E1 -24437.432,E2 -24437.432} C_VEL
LIN {X 0,Y 143.104,Z 307.471,A -85,B 0,C 180,E1 -24441.784,E2 -24441.784} C_VEL
LIN {X 0,Y 143.151,Z 307.462,A -85,B 0,C 180,E1 -24447.332,E2 -24447.332} C_VEL
LIN {X 0,Y 143.158,Z 307.465,A -85,B 0,C 180,E1 -24452.076,E2 -24452.076} C_VEL
LIN {X 0,Y 143.241,Z 307.45,A -85,B 0,C 180,E1 -24458.769,E2 -24458.769} C_VEL
LIN {X 0,Y 143.244,Z 307.453,A -85,B 0,C 180,E1 -24462.895,E2 -24462.895} C_VEL
LIN {X 0,Y 143.513,Z 307.419,A -85,B 0,C 180,E1 -24468.719,E2 -24468.719} C_VEL
LIN {X 0,Y 143.603,Z 307.409,A -85,B 0,C 180,E1 -24471.572,E2 -24471.572} C_VEL
LIN {X 0,Y 144.142,Z 307.342,A -85,B 0,C 180,E1 -24480.014,E2 -24480.014} C_VEL
LIN {X 0,Y 143.597,Z 307.41,A -85,B 0,C 180,E1 -24488.457,E2 -24488.457} C_VEL
LIN {X 0,Y 143.49,Z 307.42,A -85,B 0,C 180,E1 -24491.627,E2 -24491.627} C_VEL
LIN {X 0,Y 143.247,Z 307.455,A -85,B 0,C 180,E1 -24497.134,E2 -24497.134} C_VEL
LIN {X 0,Y 143.216,Z 307.453,A -85,B 0,C 180,E1 -24501.207,E2 -24501.207} C_VEL
LIN {X 0,Y 143.143,Z 307.466,A -85,B 0,C 180,E1 -24507.913,E2 -24507.913} C_VEL
LIN {X 0,Y 143.14,Z 307.464,A -85,B 0,C 180,E1 -24513.428,E2 -24513.428} C_VEL
LIN {X 0,Y 143.059,Z 307.471,A -85,B 0,C 180,E1 -24519.707,E2 -24519.707} C_VEL
LIN {X 0,Y 143.043,Z 307.478,A -85,B 0,C 180,E1 -24523.477,E2 -24523.477} C_VEL
LIN {X 0,Y 143.048,Z 307.477,A -85,B 0,C 180,E1 -24527.49,E2 -24527.49} C_VEL
LIN {X 0,Y 143.085,Z 307.472,A -85,B 0,C 180,E1 -24531.821,E2 -24531.821} C_VEL
LIN {X 0,Y 143.197,Z 307.456,A -85,B 0,C 180,E1 -24537.331,E2 -24537.331} C_VEL
LIN {X 0,Y 143.483,Z 307.424,A -85,B 0,C 180,E1 -24543.849,E2 -24543.849} C_VEL
LIN {X 0,Y 143.418,Z 307.432,A -85,B 0,C 180,E1 -24546.925,E2 -24546.925} C_VEL
LIN {X 0,Y 142.734,Z 307.522,A -85,B 0,C 180,E1 -24552.082,E2 -24552.082} C_VEL
LIN {X 0,Y 142.917,Z 309.919,A -85,B 0,C 180,E1 -24553.856,E2 -24553.856} C_VEL
LIN {X 0,Y 143.847,Z 332.573,A -85,B 0,C 180,E1 -24556.047,E2 -24556.047} C_VEL
LIN {X 0,Y 145.821,Z 353.438,A -85,B 0,C 180,E1 -24557.923,E2 -24557.923} C_VEL
LIN {X 0,Y 146.008,Z 387.392,A -85,B 0,C 180,E1 -24561.441,E2 -24561.441} C_VEL
LIN {X 0,Y 145.938,Z 398.905,A -85,B 0,C 180,E1 -24563.09,E2 -24563.09} C_VEL
LIN {X 0,Y 145.893,Z 409.532,A -85,B 0,C 180,E1 -24565.169,E2 -24565.169} C_VEL
LIN {X 0,Y 145.985,Z 419.278,A -85,B 0,C 180,E1 -24567.59,E2 -24567.59} C_VEL
LIN {X 0,Y 146.103,Z 428.164,A -85,B 0,C 180,E1 -24570.349,E2 -24570.349} C_VEL
LIN {X 0,Y 146.054,Z 434.36,A -85,B 0,C 180,E1 -24572.763,E2 -24572.763} C_VEL
LIN {X 0,Y 145.695,Z 438.597,A -85,B 0,C 180,E1 -24574.847,E2 -24574.847} C_VEL
LIN {X 0,Y 144.982,Z 444.396,A -85,B 0,C 180,E1 -24578.366,E2 -24578.366} C_VEL
LIN {X 0,Y 144.81,Z 449.837,A -85,B 0,C 180,E1 -24582.383,E2 -24582.383} C_VEL
LIN {X 0,Y 145.838,Z 454.699,A -85,B 0,C 180,E1 -24586.811,E2 -24586.811} C_VEL
LIN {X 0,Y 148.985,Z 459.471,A -85,B 0,C 180,E1 -24592.176,E2 -24592.176} C_VEL
LIN {X 0,Y 153.871,Z 462.53,A -85,B 0,C 180,E1 -24597.182,E2 -24597.182} C_VEL
LIN {X 0,Y 156.853,Z 463.616,A -85,B 0,C 180,E1 -24599.534,E2 -24599.534} C_VEL
LIN {X 0,Y 164.282,Z 464.529,A -85,B 0,C 180,E1 -24603.794,E2 -24603.794} C_VEL
LIN {X 0,Y 168.517,Z 464.531,A -85,B 0,C 180,E1 -24605.728,E2 -24605.728} C_VEL
LIN {X 0,Y 173.052,Z 464.025,A -85,B 0,C 180,E1 -24607.535,E2 -24607.535} C_VEL
LIN {X 0,Y 182.982,Z 461.961,A -85,B 0,C 180,E1 -24610.768,E2 -24610.768} C_VEL
LIN {X 0,Y 190.986,Z 459.274,A -85,B 0,C 180,E1 -24612.908,E2 -24612.908} C_VEL
LIN {X 0,Y 199.48,Z 455.522,A -85,B 0,C 180,E1 -24614.804,E2 -24614.804} C_VEL
LIN {X 0,Y 203.649,Z 453.337,A -85,B 0,C 180,E1 -24615.606,E2 -24615.606} C_VEL
LIN {X 0,Y 204.319,Z 452.94,A -85,B 0,C 180,E1 -24616.157,E2 -24616.157} C_VEL
LIN {X 0,Y 197.816,Z 455.906,A -85,B 0,C 180,E1 -24617.533,E2 -24617.533} C_VEL
LIN {X 0,Y 192.275,Z 457.877,A -85,B 0,C 180,E1 -24618.846,E2 -24618.846} C_VEL
LIN {X 0,Y 185.919,Z 459.605,A -85,B 0,C 180,E1 -24620.566,E2 -24620.566} C_VEL
LIN {X 0,Y 181.275,Z 460.631,A -85,B 0,C 180,E1 -24621.678,E2 -24621.678} C_VEL
LIN {X 0,Y 176.153,Z 461.373,A -85,B 0,C 180,E1 -24622.626,E2 -24622.626} C_VEL
LIN {X 0,Y 167.505,Z 461.716,A -85,B 0,C 180,E1 -24624.23,E2 -24624.23} C_VEL
LIN {X 0,Y 161.433,Z 461.181,A -85,B 0,C 180,E1 -24625.948,E2 -24625.948} C_VEL
LIN {X 0,Y 160.187,Z 460.957,A -85,B 0,C 180,E1 -24626.482,E2 -24626.482} C_VEL
LIN {X 0,Y 153.811,Z 459.056,A -85,B 0,C 180,E1 -24629.813,E2 -24629.813} C_VEL
LIN {X 0,Y 148.629,Z 456.372,A -85,B 0,C 180,E1 -24633.293,E2 -24633.293} C_VEL
LIN {X 0,Y 144.298,Z 452.71,A -85,B 0,C 180,E1 -24637.054,E2 -24637.054} C_VEL
LIN {X 0,Y 141.4,Z 448.714,A -85,B 0,C 180,E1 -24640.646,E2 -24640.646} C_VEL
LIN {X 0,Y 139.072,Z 443.509,A -85,B 0,C 180,E1 -24644.6,E2 -24644.6} C_VEL
LIN {X 0,Y 137.786,Z 436.849,A -85,B 0,C 180,E1 -24648.958,E2 -24648.958} C_VEL
LIN {X 0,Y 137.448,Z 430.283,A -85,B 0,C 180,E1 -24652.641,E2 -24652.641} C_VEL
LIN {X 0,Y 137.512,Z 422.173,A -85,B 0,C 180,E1 -24656.323,E2 -24656.323} C_VEL
LIN {X 0,Y 137.756,Z 414.319,A -85,B 0,C 180,E1 -24659.255,E2 -24659.255} C_VEL
LIN {X 0,Y 137.997,Z 404.508,A -85,B 0,C 180,E1 -24662.174,E2 -24662.174} C_VEL
LIN {X 0,Y 138.192,Z 395.184,A -85,B 0,C 180,E1 -24664.36,E2 -24664.36} C_VEL
LIN {X 0,Y 138.457,Z 385.344,A -85,B 0,C 180,E1 -24666.177,E2 -24666.177} C_VEL
LIN {X 0,Y 138.785,Z 372.977,A -85,B 0,C 180,E1 -24667.898,E2 -24667.898} C_VEL
LIN {X 0,Y 138.732,Z 321.82,A -85,B 0,C 180,E1 -24673.395,E2 -24673.395} C_VEL
LIN {X 0,Y 137.047,Z 308.226,A -85,B 0,C 180,E1 -24674.712,E2 -24674.712} C_VEL
LIN {X 0,Y 136.193,Z 308.327,A -85,B 0,C 180,E1 -24681.731,E2 -24681.731} C_VEL
LIN {X 0,Y 136.081,Z 308.345,A -85,B 0,C 180,E1 -24688.592,E2 -24688.592} C_VEL
LIN {X 0,Y 136.024,Z 308.354,A -85,B 0,C 180,E1 -24694.614,E2 -24694.614} C_VEL
LIN {X 0,Y 136.006,Z 308.351,A -85,B 0,C 180,E1 -24699.178,E2 -24699.178} C_VEL
LIN {X 0,Y 135.956,Z 308.361,A -85,B 0,C 180,E1 -24703.632,E2 -24703.632} C_VEL
LIN {X 0,Y 135.957,Z 308.358,A -85,B 0,C 180,E1 -24707.772,E2 -24707.772} C_VEL
LIN {X 0,Y 135.993,Z 308.355,A -85,B 0,C 180,E1 -24711.667,E2 -24711.667} C_VEL
LIN {X 0,Y 136.022,Z 308.352,A -85,B 0,C 180,E1 -24715.729,E2 -24715.729} C_VEL
LIN {X 0,Y 136.108,Z 308.342,A -85,B 0,C 180,E1 -24722.303,E2 -24722.303} C_VEL
LIN {X 0,Y 136.205,Z 308.326,A -85,B 0,C 180,E1 -24728.822,E2 -24728.822} C_VEL
LIN {X 0,Y 136.225,Z 308.326,A -85,B 0,C 180,E1 -24735.046,E2 -24735.046} C_VEL
LIN {X 0,Y 136.458,Z 308.297,A -85,B 0,C 180,E1 -24738.106,E2 -24738.106} C_VEL
LIN {X 0,Y 136.531,Z 308.29,A -85,B 0,C 180,E1 -24741.112,E2 -24741.112} C_VEL
LIN {X 0,Y 137.098,Z 308.221,A -85,B 0,C 180,E1 -24749.995,E2 -24749.995} C_VEL
LIN {X 0,Y 136.528,Z 308.29,A -85,B 0,C 180,E1 -24758.879,E2 -24758.879} C_VEL
LIN {X 0,Y 136.447,Z 308.298,A -85,B 0,C 180,E1 -24761.953,E2 -24761.953} C_VEL
LIN {X 0,Y 136.191,Z 308.333,A -85,B 0,C 180,E1 -24768.031,E2 -24768.031} C_VEL
LIN {X 0,Y 136.151,Z 308.332,A -85,B 0,C 180,E1 -24771.747,E2 -24771.747} C_VEL
LIN {X 0,Y 136.071,Z 308.348,A -85,B 0,C 180,E1 -24778.63,E2 -24778.63} C_VEL
LIN {X 0,Y 136.041,Z 308.35,A -85,B 0,C 180,E1 -24784.623,E2 -24784.623} C_VEL
LIN {X 0,Y 136.053,Z 308.345,A -85,B 0,C 180,E1 -24789.237,E2 -24789.237} C_VEL
LIN {X 0,Y 136.076,Z 308.347,A -85,B 0,C 180,E1 -24793.717,E2 -24793.717} C_VEL
LIN {X 0,Y 136.072,Z 308.343,A -85,B 0,C 180,E1 -24797.845,E2 -24797.845} C_VEL
LIN {X 0,Y 136.056,Z 308.348,A -85,B 0,C 180,E1 -24801.715,E2 -24801.715} C_VEL
LIN {X 0,Y 136.058,Z 308.348,A -85,B 0,C 180,E1 -24805.728,E2 -24805.728} C_VEL
LIN {X 0,Y 136.114,Z 308.342,A -85,B 0,C 180,E1 -24812.328,E2 -24812.328} C_VEL
LIN {X 0,Y 136.207,Z 308.326,A -85,B 0,C 180,E1 -24818.844,E2 -24818.844} C_VEL
LIN {X 0,Y 136.211,Z 308.326,A -85,B 0,C 180,E1 -24825.066,E2 -24825.066} C_VEL
LIN {X 0,Y 136.405,Z 308.302,A -85,B 0,C 180,E1 -24828.192,E2 -24828.192} C_VEL
LIN {X 0,Y 136.528,Z 308.29,A -85,B 0,C 180,E1 -24831.132,E2 -24831.132} C_VEL
LIN {X 0,Y 137.099,Z 308.219,A -85,B 0,C 180,E1 -24840.015,E2 -24840.015} C_VEL
LIN {X 0,Y 136.527,Z 308.292,A -85,B 0,C 180,E1 -24848.898,E2 -24848.898} C_VEL
LIN {X 0,Y 136.407,Z 308.302,A -85,B 0,C 180,E1 -24851.908,E2 -24851.908} C_VEL
LIN {X 0,Y 136.16,Z 308.336,A -85,B 0,C 180,E1 -24858.055,E2 -24858.055} C_VEL
LIN {X 0,Y 136.141,Z 308.332,A -85,B 0,C 180,E1 -24861.703,E2 -24861.703} C_VEL
LIN {X 0,Y 136.064,Z 308.347,A -85,B 0,C 180,E1 -24868.599,E2 -24868.599} C_VEL
LIN {X 0,Y 136.045,Z 308.349,A -85,B 0,C 180,E1 -24874.644,E2 -24874.644} C_VEL
LIN {X 0,Y 136.031,Z 308.349,A -85,B 0,C 180,E1 -24879.207,E2 -24879.207} C_VEL
LIN {X 0,Y 135.988,Z 308.358,A -85,B 0,C 180,E1 -24883.661,E2 -24883.661} C_VEL
LIN {X 0,Y 135.993,Z 308.354,A -85,B 0,C 180,E1 -24887.799,E2 -24887.799} C_VEL
LIN {X 0,Y 136.033,Z 308.349,A -85,B 0,C 180,E1 -24891.693,E2 -24891.693} C_VEL
LIN {X 0,Y 136.07,Z 308.348,A -85,B 0,C 180,E1 -24895.752,E2 -24895.752} C_VEL
LIN {X 0,Y 136.349,Z 308.314,A -85,B 0,C 180,E1 -24902.367,E2 -24902.367} C_VEL
LIN {X 0,Y 136.367,Z 308.312,A -85,B 0,C 180,E1 -24905.657,E2 -24905.657} C_VEL
LIN {X 0,Y 136.111,Z 308.342,A -85,B 0,C 180,E1 -24908.817,E2 -24908.817} C_VEL
LIN {X 0,Y 135.768,Z 308.506,A -85,B 0,C 180,E1 -24913.561,E2 -24913.561} C_VEL
LIN {X 0,Y 135.996,Z 309.665,A -85,B 0,C 180,E1 -24914.455,E2 -24914.455} C_VEL
LIN {X 0,Y 136.942,Z 331.585,A -85,B 0,C 180,E1 -24916.691,E2 -24916.691} C_VEL
LIN {X 0,Y 139.036,Z 352.857,A -85,B 0,C 180,E1 -24918.709,E2 -24918.709} C_VEL
LIN {X 0,Y 139.405,Z 387.063,A -85,B 0,C 180,E1 -24922.491,E2 -24922.491} C_VEL
LIN {X 0,Y 139.398,Z 398.519,A -85,B 0,C 180,E1 -24924.218,E2 -24924.218} C_VEL
LIN {X 0,Y 139.408,Z 409.108,A -85,B 0,C 180,E1 -24926.392,E2 -24926.392} C_VEL
LIN {X 0,Y 139.554,Z 417.57,A -85,B 0,C 180,E1 -24928.562,E2 -24928.562} C_VEL
LIN {X 0,Y 139.727,Z 425.516,A -85,B 0,C 180,E1 -24931.086,E2 -24931.086} C_VEL
LIN {X 0,Y 139.757,Z 431.877,A -85,B 0,C 180,E1 -24933.609,E2 -24933.609} C_VEL
LIN {X 0,Y 139.324,Z 436.29,A -85,B 0,C 180,E1 -24935.795,E2 -24935.795} C_VEL
LIN {X 0,Y 138.542,Z 443.362,A -85,B 0,C 180,E1 -24940.232,E2 -24940.232} C_VEL
LIN {X 0,Y 138.738,Z 448.974,A -85,B 0,C 180,E1 -24944.677,E2 -24944.677} C_VEL
LIN {X 0,Y 140.149,Z 453.673,A -85,B 0,C 180,E1 -24949.028,E2 -24949.028} C_VEL
LIN {X 0,Y 142.724,Z 457.38,A -85,B 0,C 180,E1 -24953.204,E2 -24953.204} C_VEL
LIN {X 0,Y 147.724,Z 461.112,A -85,B 0,C 180,E1 -24958.413,E2 -24958.413} C_VEL
LIN {X 0,Y 154.459,Z 463.28,A -85,B 0,C 180,E1 -24963.098,E2 -24963.098} C_VEL
LIN {X 0,Y 158.453,Z 463.907,A -85,B 0,C 180,E1 -24965.217,E2 -24965.217} C_VEL
LIN {X 0,Y 167.468,Z 463.994,A -85,B 0,C 180,E1 -24969.017,E2 -24969.017} C_VEL
LIN {X 0,Y 172.452,Z 463.47,A -85,B 0,C 180,E1 -24970.701,E2 -24970.701} C_VEL
LIN {X 0,Y 183.064,Z 461.253,A -85,B 0,C 180,E1 -24973.717,E2 -24973.717} C_VEL
LIN {X 0,Y 189.886,Z 459.124,A -85,B 0,C 180,E1 -24975.302,E2 -24975.302} C_VEL
LIN {X 0,Y 192.737,Z 457.96,A -85,B 0,C 180,E1 -24976.135,E2 -24976.135} C_VEL
LIN {X 0,Y 187.061,Z 459.602,A -85,B 0,C 180,E1 -24977.435,E2 -24977.435} C_VEL
LIN {X 0,Y 181.334,Z 460.861,A -85,B 0,C 180,E1 -24978.921,E2 -24978.921} C_VEL
LIN {X 0,Y 176.32,Z 461.518,A -85,B 0,C 180,E1 -24980.364,E2 -24980.364} C_VEL
LIN {X 0,Y 166.513,Z 461.775,A -85,B 0,C 180,E1 -24983.767,E2 -24983.767} C_VEL
LIN {X 0,Y 160.187,Z 460.957,A -85,B 0,C 180,E1 -24986.482,E2 -24986.482} C_VEL
LIN {X 0,Y 156.249,Z 460.102,A -85,B 0,C 180,E1 -24988.047,E2 -24988.047} C_VEL
LIN {X 0,Y 148.848,Z 457.728,A -85,B 0,C 180,E1 -24990.362,E2 -24990.362} C_VEL
LIN {X 0,Y 142.052,Z 454.497,A -85,B 0,C 180,E1 -24992.893,E2 -24992.893} C_VEL
LIN {X 0,Y 139.16,Z 452.231,A -85,B 0,C 180,E1 -24994.789,E2 -24994.789} C_VEL
LIN {X 0,Y 135.626,Z 447.575,A -85,B 0,C 180,E1 -24998.878,E2 -24998.878} C_VEL
LIN {X 0,Y 132.72,Z 441.172,A -85,B 0,C 180,E1 -25003.712,E2 -25003.712} C_VEL
LIN {X 0,Y 131.309,Z 432.517,A -85,B 0,C 180,E1 -25009.188,E2 -25009.188} C_VEL
LIN {X 0,Y 131.104,Z 425.122,A -85,B 0,C 180,E1 -25013.057,E2 -25013.057} C_VEL
LIN {X 0,Y 131.261,Z 418.095,A -85,B 0,C 180,E1 -25016.147,E2 -25016.147} C_VEL
LIN {X 0,Y 131.388,Z 411.712,A -85,B 0,C 180,E1 -25018.452,E2 -25018.452} C_VEL
LIN {X 0,Y 131.574,Z 402.728,A -85,B 0,C 180,E1 -25021.132,E2 -25021.132} C_VEL
LIN {X 0,Y 131.729,Z 393.147,A -85,B 0,C 180,E1 -25023.425,E2 -25023.425} C_VEL
LIN {X 0,Y 131.989,Z 381.367,A -85,B 0,C 180,E1 -25025.618,E2 -25025.618} C_VEL
LIN {X 0,Y 132.16,Z 366.802,A -85,B 0,C 180,E1 -25027.528,E2 -25027.528} C_VEL
LIN {X 0,Y 131.829,Z 321.473,A -85,B 0,C 180,E1 -25032.634,E2 -25032.634} C_VEL
LIN {X 0,Y 130.25,Z 309.073,A -85,B 0,C 180,E1 -25033.883,E2 -25033.883} C_VEL
LIN {X 0,Y 129.103,Z 309.209,A -85,B 0,C 180,E1 -25042.381,E2 -25042.381} C_VEL
LIN {X 0,Y 129.007,Z 309.225,A -85,B 0,C 180,E1 -25049.34,E2 -25049.34} C_VEL
LIN {X 0,Y 128.94,Z 309.235,A -85,B 0,C 180,E1 -25055.148,E2 -25055.148} C_VEL
LIN {X 0,Y 128.903,Z 309.234,A -85,B 0,C 180,E1 -25060.84,E2 -25060.84} C_VEL
LIN {X 0,Y 128.89,Z 309.242,A -85,B 0,C 180,E1 -25065.116,E2 -25065.116} C_VEL
LIN {X 0,Y 128.908,Z 309.233,A -85,B 0,C 180,E1 -25069.725,E2 -25069.725} C_VEL
LIN {X 0,Y 128.927,Z 309.239,A -85,B 0,C 180,E1 -25074.821,E2 -25074.821} C_VEL
LIN {X 0,Y 128.986,Z 309.227,A -85,B 0,C 180,E1 -25080.629,E2 -25080.629} C_VEL
LIN {X 0,Y 129.073,Z 309.213,A -85,B 0,C 180,E1 -25087.59,E2 -25087.59} C_VEL
LIN {X 0,Y 129.111,Z 309.214,A -85,B 0,C 180,E1 -25090.932,E2 -25090.932} C_VEL
LIN {X 0,Y 129.377,Z 309.177,A -85,B 0,C 180,E1 -25097.813,E2 -25097.813} C_VEL
LIN {X 0,Y 129.462,Z 309.17,A -85,B 0,C 180,E1 -25100.622,E2 -25100.622} C_VEL
LIN {X 0,Y 130.054,Z 309.099,A -85,B 0,C 180,E1 -25109.995,E2 -25109.995} C_VEL
LIN {X 0,Y 129.458,Z 309.171,A -85,B 0,C 180,E1 -25119.368,E2 -25119.368} C_VEL
LIN {X 0,Y 129.32,Z 309.182,A -85,B 0,C 180,E1 -25122.55,E2 -25122.55} C_VEL
LIN {X 0,Y 129.103,Z 309.215,A -85,B 0,C 180,E1 -25129.058,E2 -25129.058} C_VEL
LIN {X 0,Y 129.064,Z 309.214,A -85,B 0,C 180,E1 -25132.4,E2 -25132.4} C_VEL
LIN {X 0,Y 128.994,Z 309.226,A -85,B 0,C 180,E1 -25139.377,E2 -25139.377} C_VEL
LIN {X 0,Y 128.984,Z 309.231,A -85,B 0,C 180,E1 -25145.215,E2 -25145.215} C_VEL
LIN {X 0,Y 128.98,Z 309.224,A -85,B 0,C 180,E1 -25150.826,E2 -25150.826} C_VEL
LIN {X 0,Y 128.992,Z 309.23,A -85,B 0,C 180,E1 -25155.088,E2 -25155.088} C_VEL
LIN {X 0,Y 128.98,Z 309.224,A -85,B 0,C 180,E1 -25159.707,E2 -25159.707} C_VEL
LIN {X 0,Y 128.99,Z 309.229,A -85,B 0,C 180,E1 -25164.802,E2 -25164.802} C_VEL
LIN {X 0,Y 128.986,Z 309.227,A -85,B 0,C 180,E1 -25170.654,E2 -25170.654} C_VEL
LIN {X 0,Y 128.997,Z 309.228,A -85,B 0,C 180,E1 -25174.179,E2 -25174.179} C_VEL
LIN {X 0,Y 129.079,Z 309.212,A -85,B 0,C 180,E1 -25177.744,E2 -25177.744} C_VEL
LIN {X 0,Y 129.135,Z 309.209,A -85,B 0,C 180,E1 -25184.227,E2 -25184.227} C_VEL
LIN {X 0,Y 129.324,Z 309.183,A -85,B 0,C 180,E1 -25187.984,E2 -25187.984} C_VEL
LIN {X 0,Y 129.451,Z 309.173,A -85,B 0,C 180,E1 -25190.643,E2 -25190.643} C_VEL
LIN {X 0,Y 130.055,Z 309.097,A -85,B 0,C 180,E1 -25200.016,E2 -25200.016} C_VEL
LIN {X 0,Y 129.453,Z 309.172,A -85,B 0,C 180,E1 -25209.389,E2 -25209.389} C_VEL
LIN {X 0,Y 129.291,Z 309.187,A -85,B 0,C 180,E1 -25212.574,E2 -25212.574} C_VEL
LIN {X 0,Y 129.077,Z 309.219,A -85,B 0,C 180,E1 -25219.083,E2 -25219.083} C_VEL
LIN {X 0,Y 129.032,Z 309.217,A -85,B 0,C 180,E1 -25222.428,E2 -25222.428} C_VEL
LIN {X 0,Y 128.985,Z 309.227,A -85,B 0,C 180,E1 -25229.382,E2 -25229.382} C_VEL
LIN {X 0,Y 128.961,Z 309.233,A -85,B 0,C 180,E1 -25235.18,E2 -25235.18} C_VEL
LIN {X 0,Y 128.931,Z 309.229,A -85,B 0,C 180,E1 -25240.871,E2 -25240.871} C_VEL
LIN {X 0,Y 128.923,Z 309.238,A -85,B 0,C 180,E1 -25245.146,E2 -25245.146} C_VEL
LIN {X 0,Y 128.946,Z 309.228,A -85,B 0,C 180,E1 -25249.754,E2 -25249.754} C_VEL
LIN {X 0,Y 128.972,Z 309.231,A -85,B 0,C 180,E1 -25254.846,E2 -25254.846} C_VEL
LIN {X 0,Y 129.19,Z 309.203,A -85,B 0,C 180,E1 -25260.692,E2 -25260.692} C_VEL
LIN {X 0,Y 129.275,Z 309.195,A -85,B 0,C 180,E1 -25264.226,E2 -25264.226} C_VEL
LIN {X 0,Y 129.142,Z 309.208,A -85,B 0,C 180,E1 -25267.725,E2 -25267.725} C_VEL
LIN {X 0,Y 129.052,Z 309.281,A -85,B 0,C 180,E1 -25275.066,E2 -25275.066} C_VEL
LIN {X 0,Y 129.146,Z 311.67,A -85,B 0,C 180,E1 -25275.459,E2 -25275.459} C_VEL
LIN {X 0,Y 130.36,Z 334.175,A -85,B 0,C 180,E1 -25277.848,E2 -25277.848} C_VEL
LIN {X 0,Y 132.324,Z 352.714,A -85,B 0,C 180,E1 -25279.679,E2 -25279.679} C_VEL
LIN {X 0,Y 132.843,Z 386.695,A -85,B 0,C 180,E1 -25283.646,E2 -25283.646} C_VEL
LIN {X 0,Y 132.926,Z 397.054,A -85,B 0,C 180,E1 -25285.267,E2 -25285.267} C_VEL
LIN {X 0,Y 133.021,Z 408.516,A -85,B 0,C 180,E1 -25287.734,E2 -25287.734} C_VEL
LIN {X 0,Y 133.275,Z 416.826,A -85,B 0,C 180,E1 -25290.005,E2 -25290.005} C_VEL
LIN {X 0,Y 133.473,Z 423.654,A -85,B 0,C 180,E1 -25292.268,E2 -25292.268} C_VEL
LIN {X 0,Y 133.522,Z 429.352,A -85,B 0,C 180,E1 -25294.533,E2 -25294.533} C_VEL
LIN {X 0,Y 132.857,Z 435.218,A -85,B 0,C 180,E1 -25297.605,E2 -25297.605} C_VEL
LIN {X 0,Y 132.283,Z 442.07,A -85,B 0,C 180,E1 -25302.275,E2 -25302.275} C_VEL
LIN {X 0,Y 132.895,Z 447.908,A -85,B 0,C 180,E1 -25306.996,E2 -25306.996} C_VEL
LIN {X 0,Y 134.685,Z 452.473,A -85,B 0,C 180,E1 -25311.429,E2 -25311.429} C_VEL
LIN {X 0,Y 137.699,Z 456.321,A -85,B 0,C 180,E1 -25315.716,E2 -25315.716} C_VEL
LIN {X 0,Y 141.739,Z 459.273,A -85,B 0,C 180,E1 -25319.73,E2 -25319.73} C_VEL
LIN {X 0,Y 144.921,Z 460.874,A -85,B 0,C 180,E1 -25322.244,E2 -25322.244} C_VEL
LIN {X 0,Y 152.762,Z 462.916,A -85,B 0,C 180,E1 -25326.737,E2 -25326.737} C_VEL
LIN {X 0,Y 157.23,Z 463.51,A -85,B 0,C 180,E1 -25328.745,E2 -25328.745} C_VEL
LIN {X 0,Y 167.134,Z 463.454,A -85,B 0,C 180,E1 -25332.288,E2 -25332.288} C_VEL
LIN {X 0,Y 172.448,Z 462.929,A -85,B 0,C 180,E1 -25333.859,E2 -25333.859} C_VEL
LIN {X 0,Y 180.242,Z 461.458,A -85,B 0,C 180,E1 -25335.837,E2 -25335.837} C_VEL
LIN {X 0,Y 179.797,Z 461.44,A -85,B 0,C 180,E1 -25336.448,E2 -25336.448} C_VEL
LIN {X 0,Y 170.922,Z 462.255,A -85,B 0,C 180,E1 -25338.848,E2 -25338.848} C_VEL
LIN {X 0,Y 165.727,Z 462.294,A -85,B 0,C 180,E1 -25340.485,E2 -25340.485} C_VEL
LIN {X 0,Y 156.177,Z 460.979,A -85,B 0,C 180,E1 -25344.183,E2 -25344.183} C_VEL
LIN {X 0,Y 151.803,Z 459.838,A -85,B 0,C 180,E1 -25346.237,E2 -25346.237} C_VEL
LIN {X 0,Y 145.913,Z 457.288,A -85,B 0,C 180,E1 -25349.605,E2 -25349.605} C_VEL
LIN {X 0,Y 139.356,Z 452.429,A -85,B 0,C 180,E1 -25354.602,E2 -25354.602} C_VEL
LIN {X 0,Y 139.16,Z 452.231,A -85,B 0,C 180,E1 -25354.789,E2 -25354.789} C_VEL
LIN {X 0,Y 136.603,Z 449.857,A -85,B 0,C 180,E1 -25356.737,E2 -25356.737} C_VEL
LIN {X 0,Y 131.531,Z 444.809,A -85,B 0,C 180,E1 -25359.653,E2 -25359.653} C_VEL
LIN {X 0,Y 127.149,Z 439.016,A -85,B 0,C 180,E1 -25362.681,E2 -25362.681} C_VEL
LIN {X 0,Y 125.775,Z 435.46,A -85,B 0,C 180,E1 -25364.777,E2 -25364.777} C_VEL
LIN {X 0,Y 124.955,Z 427.658,A -85,B 0,C 180,E1 -25369.452,E2 -25369.452} C_VEL
LIN {X 0,Y 124.919,Z 419.3,A -85,B 0,C 180,E1 -25373.523,E2 -25373.523} C_VEL
LIN {X 0,Y 125.137,Z 412.411,A -85,B 0,C 180,E1 -25376.361,E2 -25376.361} C_VEL
LIN {X 0,Y 125.21,Z 403.838,A -85,B 0,C 180,E1 -25379.18,E2 -25379.18} C_VEL
LIN {X 0,Y 125.305,Z 394.539,A -85,B 0,C 180,E1 -25381.591,E2 -25381.591} C_VEL
LIN {X 0,Y 125.452,Z 382.671,A -85,B 0,C 180,E1 -25383.999,E2 -25383.999} C_VEL
LIN {X 0,Y 125.681,Z 368.734,A -85,B 0,C 180,E1 -25386.002,E2 -25386.002} C_VEL
LIN {X 0,Y 125.024,Z 321.422,A -85,B 0,C 180,E1 -25391.74,E2 -25391.74} C_VEL
LIN {X 0,Y 123.513,Z 309.912,A -85,B 0,C 180,E1 -25392.929,E2 -25392.929} C_VEL
LIN {X 0,Y 121.975,Z 310.098,A -85,B 0,C 180,E1 -25403.767,E2 -25403.767} C_VEL
LIN {X 0,Y 121.915,Z 310.106,A -85,B 0,C 180,E1 -25410.142,E2 -25410.142} C_VEL
LIN {X 0,Y 121.864,Z 310.118,A -85,B 0,C 180,E1 -25416.15,E2 -25416.15} C_VEL
LIN {X 0,Y 121.843,Z 310.115,A -85,B 0,C 180,E1 -25421.415,E2 -25421.415} C_VEL
LIN {X 0,Y 121.838,Z 310.115,A -85,B 0,C 180,E1 -25428.551,E2 -25428.551} C_VEL
LIN {X 0,Y 121.878,Z 310.116,A -85,B 0,C 180,E1 -25434.779,E2 -25434.779} C_VEL
LIN {X 0,Y 121.896,Z 310.11,A -85,B 0,C 180,E1 -25439.826,E2 -25439.826} C_VEL
LIN {X 0,Y 121.947,Z 310.102,A -85,B 0,C 180,E1 -25446.202,E2 -25446.202} C_VEL
LIN {X 0,Y 122.006,Z 310.098,A -85,B 0,C 180,E1 -25449.775,E2 -25449.775} C_VEL
LIN {X 0,Y 122.209,Z 310.066,A -85,B 0,C 180,E1 -25456.696,E2 -25456.696} C_VEL
LIN {X 0,Y 122.396,Z 310.052,A -85,B 0,C 180,E1 -25460.075,E2 -25460.075} C_VEL
LIN {X 0,Y 122.581,Z 310.024,A -85,B 0,C 180,E1 -25466.708,E2 -25466.708} C_VEL
LIN {X 0,Y 123.008,Z 309.976,A -85,B 0,C 180,E1 -25469.994,E2 -25469.994} C_VEL
LIN {X 0,Y 122.392,Z 310.05,A -85,B 0,C 180,E1 -25476.589,E2 -25476.589} C_VEL
LIN {X 0,Y 122.392,Z 310.052,A -85,B 0,C 180,E1 -25479.914,E2 -25479.914} C_VEL
LIN {X 0,Y 122.204,Z 310.067,A -85,B 0,C 180,E1 -25483.294,E2 -25483.294} C_VEL
LIN {X 0,Y 121.998,Z 310.099,A -85,B 0,C 180,E1 -25490.215,E2 -25490.215} C_VEL
LIN {X 0,Y 121.939,Z 310.103,A -85,B 0,C 180,E1 -25493.787,E2 -25493.787} C_VEL
LIN {X 0,Y 121.9,Z 310.109,A -85,B 0,C 180,E1 -25500.178,E2 -25500.178} C_VEL
LIN {X 0,Y 121.898,Z 310.113,A -85,B 0,C 180,E1 -25506.213,E2 -25506.213} C_VEL
LIN {X 0,Y 121.908,Z 310.106,A -85,B 0,C 180,E1 -25511.486,E2 -25511.486} C_VEL
LIN {X 0,Y 121.908,Z 310.107,A -85,B 0,C 180,E1 -25518.533,E2 -25518.533} C_VEL
LIN {X 0,Y 121.942,Z 310.107,A -85,B 0,C 180,E1 -25524.829,E2 -25524.829} C_VEL
LIN {X 0,Y 121.898,Z 310.108,A -85,B 0,C 180,E1 -25529.849,E2 -25529.849} C_VEL
LIN {X 0,Y 121.954,Z 310.1,A -85,B 0,C 180,E1 -25536.229,E2 -25536.229} C_VEL
LIN {X 0,Y 121.994,Z 310.098,A -85,B 0,C 180,E1 -25539.797,E2 -25539.797} C_VEL
LIN {X 0,Y 122.168,Z 310.072,A -85,B 0,C 180,E1 -25546.714,E2 -25546.714} C_VEL
LIN {X 0,Y 122.377,Z 310.053,A -85,B 0,C 180,E1 -25550.097,E2 -25550.097} C_VEL
LIN {X 0,Y 122.548,Z 310.027,A -85,B 0,C 180,E1 -25556.729,E2 -25556.729} C_VEL
LIN {X 0,Y 123.008,Z 309.975,A -85,B 0,C 180,E1 -25560.016,E2 -25560.016} C_VEL
LIN {X 0,Y 122.397,Z 310.048,A -85,B 0,C 180,E1 -25566.611,E2 -25566.611} C_VEL
LIN {X 0,Y 122.382,Z 310.052,A -85,B 0,C 180,E1 -25569.937,E2 -25569.937} C_VEL
LIN {X 0,Y 122.18,Z 310.07,A -85,B 0,C 180,E1 -25573.318,E2 -25573.318} C_VEL
LIN {X 0,Y 121.983,Z 310.1,A -85,B 0,C 180,E1 -25580.24,E2 -25580.24} C_VEL
LIN {X 0,Y 121.911,Z 310.108,A -85,B 0,C 180,E1 -25583.816,E2 -25583.816} C_VEL
LIN {X 0,Y 121.908,Z 310.107,A -85,B 0,C 180,E1 -25590.159,E2 -25590.159} C_VEL
LIN {X 0,Y 121.886,Z 310.114,A -85,B 0,C 180,E1 -25596.183,E2 -25596.183} C_VEL
LIN {X 0,Y 121.872,Z 310.109,A -85,B 0,C 180,E1 -25601.447,E2 -25601.447} C_VEL
LIN {X 0,Y 121.875,Z 310.109,A -85,B 0,C 180,E1 -25608.582,E2 -25608.582} C_VEL
LIN {X 0,Y 121.924,Z 310.109,A -85,B 0,C 180,E1 -25614.808,E2 -25614.808} C_VEL
LIN {X 0,Y 122.081,Z 310.084,A -85,B 0,C 180,E1 -25619.742,E2 -25619.742} C_VEL
LIN {X 0,Y 122.138,Z 310.084,A -85,B 0,C 180,E1 -25622.598,E2 -25622.598} C_VEL
LIN {X 0,Y 122.127,Z 310.082,A -85,B 0,C 180,E1 -25627.07,E2 -25627.07} C_VEL
LIN {X 0,Y 122.141,Z 310.082,A -85,B 0,C 180,E1 -25635.851,E2 -25635.851} C_VEL
LIN {X 0,Y 122.306,Z 310.255,A -85,B 0,C 180,E1 -25636.189,E2 -25636.189} C_VEL
LIN {X 0,Y 123.459,Z 331.974,A -85,B 0,C 180,E1 -25638.617,E2 -25638.617} C_VEL
LIN {X 0,Y 125.653,Z 352.49,A -85,B 0,C 180,E1 -25640.752,E2 -25640.752} C_VEL
LIN {X 0,Y 126.438,Z 386.53,A -85,B 0,C 180,E1 -25645.023,E2 -25645.023} C_VEL
LIN {X 0,Y 126.601,Z 398.154,A -85,B 0,C 180,E1 -25647.02,E2 -25647.02} C_VEL
LIN {X 0,Y 126.875,Z 409.007,A -85,B 0,C 180,E1 -25649.569,E2 -25649.569} C_VEL
LIN {X 0,Y 127.145,Z 417.163,A -85,B 0,C 180,E1 -25651.985,E2 -25651.985} C_VEL
LIN {X 0,Y 127.408,Z 424.75,A -85,B 0,C 180,E1 -25654.753,E2 -25654.753} C_VEL
LIN {X 0,Y 127.288,Z 428.278,A -85,B 0,C 180,E1 -25656.345,E2 -25656.345} C_VEL
LIN {X 0,Y 126.404,Z 436.243,A -85,B 0,C 180,E1 -25661.227,E2 -25661.227} C_VEL
LIN {X 0,Y 126.44,Z 442.734,A -85,B 0,C 180,E1 -25666.141,E2 -25666.141} C_VEL
LIN {X 0,Y 127.805,Z 447.931,A -85,B 0,C 180,E1 -25670.763,E2 -25670.763} C_VEL
LIN {X 0,Y 130.558,Z 452.629,A -85,B 0,C 180,E1 -25675.514,E2 -25675.514} C_VEL
LIN {X 0,Y 135.858,Z 457.305,A -85,B 0,C 180,E1 -25681.157,E2 -25681.157} C_VEL
LIN {X 0,Y 143.003,Z 460.594,A -85,B 0,C 180,E1 -25686.145,E2 -25686.145} C_VEL
LIN {X 0,Y 151.823,Z 462.539,A -85,B 0,C 180,E1 -25690.401,E2 -25690.401} C_VEL
LIN {X 0,Y 156.698,Z 463.079,A -85,B 0,C 180,E1 -25692.285,E2 -25692.285} C_VEL
LIN {X 0,Y 168.329,Z 462.836,A -85,B 0,C 180,E1 -25695.807,E2 -25695.807} C_VEL
LIN {X 0,Y 167.48,Z 462.751,A -85,B 0,C 180,E1 -25696.705,E2 -25696.705} C_VEL
LIN {X 0,Y 160.305,Z 462.34,A -85,B 0,C 180,E1 -25698.867,E2 -25698.867} C_VEL
LIN {X 0,Y 150.487,Z 460.513,A -85,B 0,C 180,E1 -25702.604,E2 -25702.604} C_VEL
LIN {X 0,Y 141.832,Z 457.045,A -85,B 0,C 180,E1 -25706.956,E2 -25706.956} C_VEL
LIN {X 0,Y 136.369,Z 453.464,A -85,B 0,C 180,E1 -25710.671,E2 -25710.671} C_VEL
LIN {X 0,Y 131.834,Z 448.949,A -85,B 0,C 180,E1 -25714.74,E2 -25714.74} C_VEL
LIN {X 0,Y 128.927,Z 444.528,A -85,B 0,C 180,E1 -25718.395,E2 -25718.395} C_VEL
LIN {X 0,Y 126.101,Z 436.899,A -85,B 0,C 180,E1 -25723.804,E2 -25723.804} C_VEL
LIN {X 0,Y 125.775,Z 435.46,A -85,B 0,C 180,E1 -25724.777,E2 -25724.777} C_VEL
LIN {X 0,Y 124.705,Z 431.787,A -85,B 0,C 180,E1 -25726.836,E2 -25726.836} C_VEL
LIN {X 0,Y 123.084,Z 427.678,A -85,B 0,C 180,E1 -25728.644,E2 -25728.644} C_VEL
LIN {X 0,Y 119.796,Z 418.434,A -85,B 0,C 180,E1 -25731.956,E2 -25731.956} C_VEL
LIN {X 0,Y 118.985,Z 413.732,A -85,B 0,C 180,E1 -25733.674,E2 -25733.674} C_VEL
LIN {X 0,Y 118.958,Z 412.132,A -85,B 0,C 180,E1 -25734.273,E2 -25734.273} C_VEL
LIN {X 0,Y 119.03,Z 403.079,A -85,B 0,C 180,E1 -25737.445,E2 -25737.445} C_VEL
LIN {X 0,Y 119.011,Z 392.267,A -85,B 0,C 180,E1 -25740.406,E2 -25740.406} C_VEL
LIN {X 0,Y 119.093,Z 381.543,A -85,B 0,C 180,E1 -25742.625,E2 -25742.625} C_VEL
LIN {X 0,Y 119.241,Z 368.208,A -85,B 0,C 180,E1 -25744.631,E2 -25744.631} C_VEL
LIN {X 0,Y 118.254,Z 321.063,A -85,B 0,C 180,E1 -25750.685,E2 -25750.685} C_VEL
LIN {X 0,Y 116.863,Z 310.743,A -85,B 0,C 180,E1 -25751.802,E2 -25751.802} C_VEL
LIN {X 0,Y 114.941,Z 310.973,A -85,B 0,C 180,E1 -25763.471,E2 -25763.471} C_VEL
LIN {X 0,Y 114.843,Z 310.984,A -85,B 0,C 180,E1 -25771.036,E2 -25771.036} C_VEL
LIN {X 0,Y 114.757,Z 311.001,A -85,B 0,C 180,E1 -25777.74,E2 -25777.74} C_VEL
LIN {X 0,Y 114.757,Z 311,A -85,B 0,C 180,E1 -25782.693,E2 -25782.693} C_VEL
LIN {X 0,Y 114.762,Z 310.998,A -85,B 0,C 180,E1 -25787.644,E2 -25787.644} C_VEL
LIN {X 0,Y 114.756,Z 311.002,A -85,B 0,C 180,E1 -25792.731,E2 -25792.731} C_VEL
LIN {X 0,Y 114.824,Z 310.987,A -85,B 0,C 180,E1 -25798.93,E2 -25798.93} C_VEL
LIN {X 0,Y 114.912,Z 310.978,A -85,B 0,C 180,E1 -25806.496,E2 -25806.496} C_VEL
LIN {X 0,Y 114.971,Z 310.976,A -85,B 0,C 180,E1 -25812.197,E2 -25812.197} C_VEL
LIN {X 0,Y 115.224,Z 310.937,A -85,B 0,C 180,E1 -25817.303,E2 -25817.303} C_VEL
LIN {X 0,Y 115.338,Z 310.928,A -85,B 0,C 180,E1 -25822.994,E2 -25822.994} C_VEL
LIN {X 0,Y 115.961,Z 310.854,A -85,B 0,C 180,E1 -25829.994,E2 -25829.994} C_VEL
LIN {X 0,Y 115.335,Z 310.929,A -85,B 0,C 180,E1 -25836.994,E2 -25836.994} C_VEL
LIN {X 0,Y 115.218,Z 310.938,A -85,B 0,C 180,E1 -25842.685,E2 -25842.685} C_VEL
LIN {X 0,Y 114.963,Z 310.977,A -85,B 0,C 180,E1 -25847.792,E2 -25847.792} C_VEL
LIN {X 0,Y 114.902,Z 310.979,A -85,B 0,C 180,E1 -25853.492,E2 -25853.492} C_VEL
LIN {X 0,Y 114.827,Z 310.986,A -85,B 0,C 180,E1 -25861.073,E2 -25861.073} C_VEL
LIN {X 0,Y 114.81,Z 310.994,A -85,B 0,C 180,E1 -25867.736,E2 -25867.736} C_VEL
LIN {X 0,Y 114.831,Z 310.99,A -85,B 0,C 180,E1 -25872.77,E2 -25872.77} C_VEL
LIN {X 0,Y 114.835,Z 310.988,A -85,B 0,C 180,E1 -25877.712,E2 -25877.712} C_VEL
LIN {X 0,Y 114.821,Z 310.993,A -85,B 0,C 180,E1 -25882.711,E2 -25882.711} C_VEL
LIN {X 0,Y 114.832,Z 310.985,A -85,B 0,C 180,E1 -25888.95,E2 -25888.95} C_VEL
LIN {X 0,Y 114.919,Z 310.976,A -85,B 0,C 180,E1 -25896.524,E2 -25896.524} C_VEL
LIN {X 0,Y 114.96,Z 310.978,A -85,B 0,C 180,E1 -25902.221,E2 -25902.221} C_VEL
LIN {X 0,Y 115.289,Z 310.935,A -85,B 0,C 180,E1 -25909.481,E2 -25909.481} C_VEL
LIN {X 0,Y 115.475,Z 310.907,A -85,B 0,C 180,E1 -25916.528,E2 -25916.528} C_VEL
LIN {X 0,Y 115.96,Z 310.853,A -85,B 0,C 180,E1 -25920.017,E2 -25920.017} C_VEL
LIN {X 0,Y 115.339,Z 310.929,A -85,B 0,C 180,E1 -25927.017,E2 -25927.017} C_VEL
LIN {X 0,Y 115.197,Z 310.942,A -85,B 0,C 180,E1 -25932.574,E2 -25932.574} C_VEL
LIN {X 0,Y 114.959,Z 310.977,A -85,B 0,C 180,E1 -25937.816,E2 -25937.816} C_VEL
LIN {X 0,Y 114.892,Z 310.98,A -85,B 0,C 180,E1 -25943.446,E2 -25943.446} C_VEL
LIN {X 0,Y 114.844,Z 310.985,A -85,B 0,C 180,E1 -25951.06,E2 -25951.06} C_VEL
LIN {X 0,Y 114.781,Z 310.998,A -85,B 0,C 180,E1 -25957.775,E2 -25957.775} C_VEL
LIN {X 0,Y 114.788,Z 310.996,A -85,B 0,C 180,E1 -25962.727,E2 -25962.727} C_VEL
LIN {X 0,Y 114.798,Z 310.994,A -85,B 0,C 180,E1 -25967.677,E2 -25967.677} C_VEL
LIN {X 0,Y 114.798,Z 310.997,A -85,B 0,C 180,E1 -25972.762,E2 -25972.762} C_VEL
LIN {X 0,Y 114.976,Z 310.968,A -85,B 0,C 180,E1 -25978.873,E2 -25978.873} C_VEL
LIN {X 0,Y 115.03,Z 310.969,A -85,B 0,C 180,E1 -25984.687,E2 -25984.687} C_VEL
LIN {X 0,Y 114.863,Z 310.987,A -85,B 0,C 180,E1 -25988.469,E2 -25988.469} C_VEL
LIN {X 0,Y 115.536,Z 310.903,A -85,B 0,C 180,E1 -25997.283,E2 -25997.283} C_VEL
LIN {X 0,Y 117.018,Z 333.952,A -85,B 0,C 180,E1 -26000.063,E2 -26000.063} C_VEL
LIN {X 0,Y 119.121,Z 352.239,A -85,B 0,C 180,E1 -26002.058,E2 -26002.058} C_VEL
LIN {X 0,Y 120.127,Z 384.786,A -85,B 0,C 180,E1 -26006.34,E2 -26006.34} C_VEL
LIN {X 0,Y 120.366,Z 395.296,A -85,B 0,C 180,E1 -26008.165,E2 -26008.165} C_VEL
LIN {X 0,Y 120.619,Z 406.009,A -85,B 0,C 180,E1 -26010.632,E2 -26010.632} C_VEL
LIN {X 0,Y 121.039,Z 414.983,A -85,B 0,C 180,E1 -26013.334,E2 -26013.334} C_VEL
LIN {X 0,Y 121.426,Z 422.271,A -85,B 0,C 180,E1 -26016.078,E2 -26016.078} C_VEL
LIN {X 0,Y 121.171,Z 426.806,A -85,B 0,C 180,E1 -26018.345,E2 -26018.345} C_VEL
LIN {X 0,Y 120.347,Z 434.805,A -85,B 0,C 180,E1 -26023.514,E2 -26023.514} C_VEL
LIN {X 0,Y 120.973,Z 441.683,A -85,B 0,C 180,E1 -26029.055,E2 -26029.055} C_VEL
LIN {X 0,Y 122.708,Z 446.718,A -85,B 0,C 180,E1 -26033.641,E2 -26033.641} C_VEL
LIN {X 0,Y 125.905,Z 451.253,A -85,B 0,C 180,E1 -26038.33,E2 -26038.33} C_VEL
LIN {X 0,Y 130.168,Z 455.008,A -85,B 0,C 180,E1 -26042.684,E2 -26042.684} C_VEL
LIN {X 0,Y 133.572,Z 457.078,A -85,B 0,C 180,E1 -26045.37,E2 -26045.37} C_VEL
LIN {X 0,Y 141.847,Z 460.263,A -85,B 0,C 180,E1 -26050.104,E2 -26050.104} C_VEL
LIN {X 0,Y 151.58,Z 462.108,A -85,B 0,C 180,E1 -26054.07,E2 -26054.07} C_VEL
LIN {X 0,Y 156.935,Z 462.635,A -85,B 0,C 180,E1 -26055.774,E2 -26055.774} C_VEL
LIN {X 0,Y 155.021,Z 462.209,A -85,B 0,C 180,E1 -26057.139,E2 -26057.139} C_VEL
LIN {X 0,Y 149.846,Z 461.114,A -85,B 0,C 180,E1 -26058.942,E2 -26058.942} C_VEL
LIN {X 0,Y 140.313,Z 457.851,A -85,B 0,C 180,E1 -26063.039,E2 -26063.039} C_VEL
LIN {X 0,Y 134.105,Z 454.388,A -85,B 0,C 180,E1 -26066.598,E2 -26066.598} C_VEL
LIN {X 0,Y 128.711,Z 450.057,A -85,B 0,C 180,E1 -26070.55,E2 -26070.55} C_VEL
LIN {X 0,Y 124.379,Z 444.544,A -85,B 0,C 180,E1 -26075.126,E2 -26075.126} C_VEL
LIN {X 0,Y 121.333,Z 438.517,A -85,B 0,C 180,E1 -26079.647,E2 -26079.647} C_VEL
LIN {X 0,Y 119.53,Z 431.016,A -85,B 0,C 180,E1 -26084.641,E2 -26084.641} C_VEL
LIN {X 0,Y 118.854,Z 422.171,A -85,B 0,C 180,E1 -26089.765,E2 -26089.765} C_VEL
LIN {X 0,Y 118.958,Z 412.132,A -85,B 0,C 180,E1 -26094.273,E2 -26094.273} C_VEL
LIN {X 0,Y 118.477,Z 407.475,A -85,B 0,C 180,E1 -26095.846,E2 -26095.846} C_VEL
LIN {X 0,Y 117.23,Z 402.424,A -85,B 0,C 180,E1 -26097.066,E2 -26097.066} C_VEL
LIN {X 0,Y 114.035,Z 391.476,A -85,B 0,C 180,E1 -26099.007,E2 -26099.007} C_VEL
LIN {X 0,Y 113.06,Z 385.553,A -85,B 0,C 180,E1 -26100.015,E2 -26100.015} C_VEL
LIN {X 0,Y 112.952,Z 383.591,A -85,B 0,C 180,E1 -26100.402,E2 -26100.402} C_VEL
LIN {X 0,Y 112.967,Z 369.526,A -85,B 0,C 180,E1 -26102.768,E2 -26102.768} C_VEL
LIN {X 0,Y 111.721,Z 321.771,A -85,B 0,C 180,E1 -26109.372,E2 -26109.372} C_VEL
LIN {X 0,Y 110.284,Z 311.564,A -85,B 0,C 180,E1 -26110.538,E2 -26110.538} C_VEL
LIN {X 0,Y 108.101,Z 311.831,A -85,B 0,C 180,E1 -26118.949,E2 -26118.949} C_VEL
LIN {X 0,Y 107.849,Z 311.858,A -85,B 0,C 180,E1 -26124.16,E2 -26124.16} C_VEL
LIN {X 0,Y 107.765,Z 311.865,A -85,B 0,C 180,E1 -26132.016,E2 -26132.016} C_VEL
LIN {X 0,Y 107.665,Z 311.883,A -85,B 0,C 180,E1 -26138.425,E2 -26138.425} C_VEL
LIN {X 0,Y 107.647,Z 311.888,A -85,B 0,C 180,E1 -26145.873,E2 -26145.873} C_VEL
LIN {X 0,Y 107.656,Z 311.885,A -85,B 0,C 180,E1 -26151.537,E2 -26151.537} C_VEL
LIN {X 0,Y 107.76,Z 311.866,A -85,B 0,C 180,E1 -26158.543,E2 -26158.543} C_VEL
LIN {X 0,Y 107.876,Z 311.853,A -85,B 0,C 180,E1 -26166.983,E2 -26166.983} C_VEL
LIN {X 0,Y 107.994,Z 311.841,A -85,B 0,C 180,E1 -26174.905,E2 -26174.905} C_VEL
LIN {X 0,Y 108.231,Z 311.813,A -85,B 0,C 180,E1 -26178.76,E2 -26178.76} C_VEL
LIN {X 0,Y 108.426,Z 311.785,A -85,B 0,C 180,E1 -26186.277,E2 -26186.277} C_VEL
LIN {X 0,Y 108.911,Z 311.732,A -85,B 0,C 180,E1 -26189.994,E2 -26189.994} C_VEL
LIN {X 0,Y 108.274,Z 311.808,A -85,B 0,C 180,E1 -26197.453,E2 -26197.453} C_VEL
LIN {X 0,Y 108.139,Z 311.819,A -85,B 0,C 180,E1 -26202.973,E2 -26202.973} C_VEL
LIN {X 0,Y 107.857,Z 311.861,A -85,B 0,C 180,E1 -26209.007,E2 -26209.007} C_VEL
LIN {X 0,Y 107.814,Z 311.863,A -85,B 0,C 180,E1 -26214.185,E2 -26214.185} C_VEL
LIN {X 0,Y 107.758,Z 311.867,A -85,B 0,C 180,E1 -26222.061,E2 -26222.061} C_VEL
LIN {X 0,Y 107.717,Z 311.877,A -85,B 0,C 180,E1 -26228.504,E2 -26228.504} C_VEL
LIN {X 0,Y 107.734,Z 311.877,A -85,B 0,C 180,E1 -26235.845,E2 -26235.845} C_VEL
LIN {X 0,Y 107.721,Z 311.876,A -85,B 0,C 180,E1 -26241.517,E2 -26241.517} C_VEL
LIN {X 0,Y 107.775,Z 311.863,A -85,B 0,C 180,E1 -26248.579,E2 -26248.579} C_VEL
LIN {X 0,Y 107.881,Z 311.852,A -85,B 0,C 180,E1 -26257.013,E2 -26257.013} C_VEL
LIN {X 0,Y 107.962,Z 311.845,A -85,B 0,C 180,E1 -26264.927,E2 -26264.927} C_VEL
LIN {X 0,Y 108.206,Z 311.817,A -85,B 0,C 180,E1 -26268.784,E2 -26268.784} C_VEL
LIN {X 0,Y 108.275,Z 311.809,A -85,B 0,C 180,E1 -26272.56,E2 -26272.56} C_VEL
LIN {X 0,Y 108.886,Z 311.734,A -85,B 0,C 180,E1 -26280.019,E2 -26280.019} C_VEL
LIN {X 0,Y 108.278,Z 311.809,A -85,B 0,C 180,E1 -26287.477,E2 -26287.477} C_VEL
LIN {X 0,Y 108.131,Z 311.82,A -85,B 0,C 180,E1 -26292.89,E2 -26292.89} C_VEL
LIN {X 0,Y 107.857,Z 311.862,A -85,B 0,C 180,E1 -26299.033,E2 -26299.033} C_VEL
LIN {X 0,Y 107.801,Z 311.865,A -85,B 0,C 180,E1 -26304.134,E2 -26304.134} C_VEL
LIN {X 0,Y 107.772,Z 311.866,A -85,B 0,C 180,E1 -26312.045,E2 -26312.045} C_VEL
LIN {X 0,Y 107.69,Z 311.88,A -85,B 0,C 180,E1 -26318.463,E2 -26318.463} C_VEL
LIN {X 0,Y 107.681,Z 311.884,A -85,B 0,C 180,E1 -26325.908,E2 -26325.908} C_VEL
LIN {X 0,Y 107.697,Z 311.878,A -85,B 0,C 180,E1 -26331.57,E2 -26331.57} C_VEL
LIN {X 0,Y 107.915,Z 311.847,A -85,B 0,C 180,E1 -26338.608,E2 -26338.608} C_VEL
LIN {X 0,Y 108.005,Z 311.843,A -85,B 0,C 180,E1 -26345.681,E2 -26345.681} C_VEL
LIN {X 0,Y 108.71,Z 311.757,A -85,B 0,C 180,E1 -26358.286,E2 -26358.286} C_VEL
LIN {X 0,Y 108.93,Z 311.727,A -85,B 0,C 180,E1 -26358.645,E2 -26358.645} C_VEL
LIN {X 0,Y 110.525,Z 334.25,A -85,B 0,C 180,E1 -26361.493,E2 -26361.493} C_VEL
LIN {X 0,Y 112.665,Z 351.829,A -85,B 0,C 180,E1 -26363.502,E2 -26363.502} C_VEL
LIN {X 0,Y 113.923,Z 384.043,A -85,B 0,C 180,E1 -26367.989,E2 -26367.989} C_VEL
LIN {X 0,Y 114.284,Z 393.89,A -85,B 0,C 180,E1 -26369.792,E2 -26369.792} C_VEL
LIN {X 0,Y 114.666,Z 403.847,A -85,B 0,C 180,E1 -26372.201,E2 -26372.201} C_VEL
LIN {X 0,Y 115.209,Z 413.673,A -85,B 0,C 180,E1 -26375.227,E2 -26375.227} C_VEL
LIN {X 0,Y 115.589,Z 420.4,A -85,B 0,C 180,E1 -26377.87,E2 -26377.87} C_VEL
LIN {X 0,Y 115.047,Z 426.294,A -85,B 0,C 180,E1 -26381.189,E2 -26381.189} C_VEL
LIN {X 0,Y 114.81,Z 435.347,A -85,B 0,C 180,E1 -26387.829,E2 -26387.829} C_VEL
LIN {X 0,Y 115.923,Z 440.822,A -85,B 0,C 180,E1 -26392.493,E2 -26392.493} C_VEL
LIN {X 0,Y 119.033,Z 446.754,A -85,B 0,C 180,E1 -26398.192,E2 -26398.192} C_VEL
LIN {X 0,Y 123.09,Z 451.143,A -85,B 0,C 180,E1 -26402.854,E2 -26402.854} C_VEL
LIN {X 0,Y 128.173,Z 454.707,A -85,B 0,C 180,E1 -26407.102,E2 -26407.102} C_VEL
LIN {X 0,Y 132.216,Z 456.821,A -85,B 0,C 180,E1 -26409.639,E2 -26409.639} C_VEL
LIN {X 0,Y 141.515,Z 459.862,A -85,B 0,C 180,E1 -26414.055,E2 -26414.055} C_VEL
LIN {X 0,Y 146.62,Z 460.973,A -85,B 0,C 180,E1 -26415.978,E2 -26415.978} C_VEL
LIN {X 0,Y 144.592,Z 460.264,A -85,B 0,C 180,E1 -26417.103,E2 -26417.103} C_VEL
LIN {X 0,Y 139.065,Z 458.34,A -85,B 0,C 180,E1 -26419.3,E2 -26419.3} C_VEL
LIN {X 0,Y 132.572,Z 455.229,A -85,B 0,C 180,E1 -26422.42,E2 -26422.42} C_VEL
LIN {X 0,Y 124.652,Z 449.345,A -85,B 0,C 180,E1 -26427.597,E2 -26427.597} C_VEL
LIN {X 0,Y 119.909,Z 444.007,A -85,B 0,C 180,E1 -26432.021,E2 -26432.021} C_VEL
LIN {X 0,Y 116.313,Z 437.579,A -85,B 0,C 180,E1 -26436.857,E2 -26436.857} C_VEL
LIN {X 0,Y 113.736,Z 428.762,A -85,B 0,C 180,E1 -26442.914,E2 -26442.914} C_VEL
LIN {X 0,Y 113.038,Z 419.359,A -85,B 0,C 180,E1 -26448.325,E2 -26448.325} C_VEL
LIN {X 0,Y 112.965,Z 410.782,A -85,B 0,C 180,E1 -26452.385,E2 -26452.385} C_VEL
LIN {X 0,Y 112.932,Z 403.691,A -85,B 0,C 180,E1 -26455.027,E2 -26455.027} C_VEL
LIN {X 0,Y 112.966,Z 396.373,A -85,B 0,C 180,E1 -26457.308,E2 -26457.308} C_VEL
LIN {X 0,Y 112.96,Z 385.517,A -85,B 0,C 180,E1 -26459.982,E2 -26459.982} C_VEL
LIN {X 0,Y 112.952,Z 383.591,A -85,B 0,C 180,E1 -26460.402,E2 -26460.402} C_VEL
LIN {X 0,Y 112.289,Z 378,A -85,B 0,C 180,E1 -26461.296,E2 -26461.296} C_VEL
LIN {X 0,Y 109.706,Z 368.537,A -85,B 0,C 180,E1 -26462.053,E2 -26462.053} C_VEL
LIN {X 0,Y 107.446,Z 360.88,A -85,B 0,C 180,E1 -26462.49,E2 -26462.49} C_VEL
LIN {X 0,Y 106.334,Z 355.09,A -85,B 0,C 180,E1 -26463.02,E2 -26463.02} C_VEL
LIN {X 0,Y 106.169,Z 353.16,A -85,B 0,C 180,E1 -26463.272,E2 -26463.272} C_VEL
LIN {X 0,Y 104.972,Z 320.439,A -85,B 0,C 180,E1 -26468.038,E2 -26468.038} C_VEL
LIN {X 0,Y 103.818,Z 312.368,A -85,B 0,C 180,E1 -26468.986,E2 -26468.986} C_VEL
LIN {X 0,Y 101.406,Z 312.665,A -85,B 0,C 180,E1 -26476.073,E2 -26476.073} C_VEL
LIN {X 0,Y 100.769,Z 312.743,A -85,B 0,C 180,E1 -26484.936,E2 -26484.936} C_VEL
LIN {X 0,Y 100.674,Z 312.753,A -85,B 0,C 180,E1 -26493.09,E2 -26493.09} C_VEL
LIN {X 0,Y 100.616,Z 312.757,A -85,B 0,C 180,E1 -26499.785,E2 -26499.785} C_VEL
LIN {X 0,Y 100.618,Z 312.763,A -85,B 0,C 180,E1 -26505.686,E2 -26505.686} C_VEL
LIN {X 0,Y 100.595,Z 312.761,A -85,B 0,C 180,E1 -26511.032,E2 -26511.032} C_VEL
LIN {X 0,Y 100.659,Z 312.754,A -85,B 0,C 180,E1 -26516.871,E2 -26516.871} C_VEL
LIN {X 0,Y 100.755,Z 312.744,A -85,B 0,C 180,E1 -26525.252,E2 -26525.252} C_VEL
LIN {X 0,Y 100.779,Z 312.74,A -85,B 0,C 180,E1 -26529.586,E2 -26529.586} C_VEL
LIN {X 0,Y 101.132,Z 312.694,A -85,B 0,C 180,E1 -26537.96,E2 -26537.96} C_VEL
LIN {X 0,Y 101.216,Z 312.689,A -85,B 0,C 180,E1 -26542.011,E2 -26542.011} C_VEL
LIN {X 0,Y 101.835,Z 312.614,A -85,B 0,C 180,E1 -26549.993,E2 -26549.993} C_VEL
LIN {X 0,Y 101.213,Z 312.689,A -85,B 0,C 180,E1 -26557.976,E2 -26557.976} C_VEL
LIN {X 0,Y 101.067,Z 312.699,A -85,B 0,C 180,E1 -26563.313,E2 -26563.313} C_VEL
LIN {X 0,Y 100.77,Z 312.742,A -85,B 0,C 180,E1 -26570.401,E2 -26570.401} C_VEL
LIN {X 0,Y 100.733,Z 312.747,A -85,B 0,C 180,E1 -26574.962,E2 -26574.962} C_VEL
LIN {X 0,Y 100.667,Z 312.753,A -85,B 0,C 180,E1 -26583.136,E2 -26583.136} C_VEL
